//   (this object) <-> Device 1 (EtherCAT)/Term 1 (EK1200)/Term 5 (EK1122)/EK1100_ST1K2_ZOS/ST1K1-EL5042
//     Enc/Inputs/In/nComState @bit 1 <-> WcState/InputToggle
//     Enc/Inputs/In/nComState <-> WcState/WcState
//     Enc/Inputs/In/nDataIn1 <-> FB Inputs Channel 1/Position
//     Enc/Inputs/In/nState1 @bit 12 <-> FB Inputs Channel 1/Status/Diag
//     Enc/Inputs/In/nState1 @bit 1 <-> FB Inputs Channel 1/Status/Error
//     Enc/Inputs/In/nState1 @bit 14 <-> FB Inputs Channel 1/Status/Input cycle counter
//     Enc/Inputs/In/nState1 @bit 2 <-> FB Inputs Channel 1/Status/Ready
//     Enc/Inputs/In/nState1 @bit 13 <-> FB Inputs Channel 1/Status/TxPDO State
//     Enc/Inputs/In/nState1 <-> FB Inputs Channel 1/Status/Warning
//   (this object) <-> Device 1 (EtherCAT)/Term 1 (EK1200)/Term 5 (EK1122)/EK1100_ST1K2_ZOS/ST1K1-EL7041
//     Drive/Inputs/In/nState1 @bit 3 <-> STM Status/Status/Error
//     Drive/Inputs/In/nState1 @bit 5 <-> STM Status/Status/Moving negative
//     Drive/Inputs/In/nState1 @bit 4 <-> STM Status/Status/Moving positive
//     Drive/Inputs/In/nState1 @bit 1 <-> STM Status/Status/Ready
//     Drive/Inputs/In/nState1 <-> STM Status/Status/Ready to enable
//     Drive/Inputs/In/nState1 @bit 6 <-> STM Status/Status/Torque reduced
//     Drive/Inputs/In/nState1 @bit 2 <-> STM Status/Status/Warning
//     Drive/Inputs/In/nState2 @bit 3 <-> STM Status/Status/Digital input 1
//     Drive/Inputs/In/nState2 @bit 4 <-> STM Status/Status/Digital input 2
//     Drive/Inputs/In/nState2 @bit 5 <-> STM Status/Status/Sync error
//     Drive/Inputs/In/nState2 @bit 7 <-> STM Status/Status/TxPDO Toggle
//     Drive/Inputs/In/nState4 @bit 1 <-> WcState/InputToggle
//     Drive/Inputs/In/nState4 <-> WcState/WcState
//     Drive/Outputs/Out/nCtrl1 <-> STM Control/Control/Enable
//     Drive/Outputs/Out/nCtrl1 @bit 2 <-> STM Control/Control/Reduce torque
//     Drive/Outputs/Out/nCtrl1 @bit 1 <-> STM Control/Control/Reset
//     Drive/Outputs/Out/nDataOut2[0] <-> STM Velocity/Velocity
//   (this object) <-> Device 1 (EtherCAT)/Term 1 (EK1200)/Term 79 (EK1521-0010)/Term 306 (EK1501-0010)/Term 310 (EK1122)/EK1100_MR2K2/EL5042_M2K2X_M2K2Y
//     Enc/Inputs/In/nComState @bit 1 <-> WcState/InputToggle
//     Enc/Inputs/In/nComState <-> WcState/WcState
//     Enc/Inputs/In/nDataIn1 <-> FB Inputs Channel 1/Position
//     Enc/Inputs/In/nDataIn1 <-> FB Inputs Channel 2/Position
//     Enc/Inputs/In/nState1 @bit 12 <-> FB Inputs Channel 1/Status/Diag
//     Enc/Inputs/In/nState1 @bit 12 <-> FB Inputs Channel 2/Status/Diag
//     Enc/Inputs/In/nState1 @bit 1 <-> FB Inputs Channel 1/Status/Error
//     Enc/Inputs/In/nState1 @bit 1 <-> FB Inputs Channel 2/Status/Error
//     Enc/Inputs/In/nState1 @bit 14 <-> FB Inputs Channel 1/Status/Input cycle counter
//     Enc/Inputs/In/nState1 @bit 14 <-> FB Inputs Channel 2/Status/Input cycle counter
//     Enc/Inputs/In/nState1 @bit 2 <-> FB Inputs Channel 1/Status/Ready
//     Enc/Inputs/In/nState1 @bit 2 <-> FB Inputs Channel 2/Status/Ready
//     Enc/Inputs/In/nState1 @bit 13 <-> FB Inputs Channel 1/Status/TxPDO State
//     Enc/Inputs/In/nState1 @bit 13 <-> FB Inputs Channel 2/Status/TxPDO State
//     Enc/Inputs/In/nState1 <-> FB Inputs Channel 1/Status/Warning
//     Enc/Inputs/In/nState1 <-> FB Inputs Channel 2/Status/Warning
//   (this object) <-> Device 1 (EtherCAT)/Term 1 (EK1200)/Term 79 (EK1521-0010)/Term 306 (EK1501-0010)/Term 310 (EK1122)/EK1100_MR2K2/EL7041_M2K2X
//     Drive/Inputs/In/nState1 @bit 3 <-> STM Status/Status/Error
//     Drive/Inputs/In/nState1 @bit 5 <-> STM Status/Status/Moving negative
//     Drive/Inputs/In/nState1 @bit 4 <-> STM Status/Status/Moving positive
//     Drive/Inputs/In/nState1 @bit 1 <-> STM Status/Status/Ready
//     Drive/Inputs/In/nState1 <-> STM Status/Status/Ready to enable
//     Drive/Inputs/In/nState1 @bit 6 <-> STM Status/Status/Torque reduced
//     Drive/Inputs/In/nState1 @bit 2 <-> STM Status/Status/Warning
//     Drive/Inputs/In/nState2 @bit 3 <-> STM Status/Status/Digital input 1
//     Drive/Inputs/In/nState2 @bit 4 <-> STM Status/Status/Digital input 2
//     Drive/Inputs/In/nState2 @bit 5 <-> STM Status/Status/Sync error
//     Drive/Inputs/In/nState2 @bit 7 <-> STM Status/Status/TxPDO Toggle
//     Drive/Inputs/In/nState4 @bit 1 <-> WcState/InputToggle
//     Drive/Inputs/In/nState4 <-> WcState/WcState
//     Drive/Outputs/Out/nCtrl1 <-> STM Control/Control/Enable
//     Drive/Outputs/Out/nCtrl1 @bit 2 <-> STM Control/Control/Reduce torque
//     Drive/Outputs/Out/nCtrl1 @bit 1 <-> STM Control/Control/Reset
//     Drive/Outputs/Out/nDataOut2[0] <-> STM Velocity/Velocity
//   (this object) <-> Device 1 (EtherCAT)/Term 1 (EK1200)/Term 79 (EK1521-0010)/Term 306 (EK1501-0010)/Term 310 (EK1122)/EK1100_MR2K2/EL7041_M2K2Y
//     Drive/Inputs/In/nState1 @bit 3 <-> STM Status/Status/Error
//     Drive/Inputs/In/nState1 @bit 5 <-> STM Status/Status/Moving negative
//     Drive/Inputs/In/nState1 @bit 4 <-> STM Status/Status/Moving positive
//     Drive/Inputs/In/nState1 @bit 1 <-> STM Status/Status/Ready
//     Drive/Inputs/In/nState1 <-> STM Status/Status/Ready to enable
//     Drive/Inputs/In/nState1 @bit 6 <-> STM Status/Status/Torque reduced
//     Drive/Inputs/In/nState1 @bit 2 <-> STM Status/Status/Warning
//     Drive/Inputs/In/nState2 @bit 3 <-> STM Status/Status/Digital input 1
//     Drive/Inputs/In/nState2 @bit 4 <-> STM Status/Status/Digital input 2
//     Drive/Inputs/In/nState2 @bit 5 <-> STM Status/Status/Sync error
//     Drive/Inputs/In/nState2 @bit 7 <-> STM Status/Status/TxPDO Toggle
//     Drive/Inputs/In/nState4 @bit 1 <-> WcState/InputToggle
//     Drive/Inputs/In/nState4 <-> WcState/WcState
//     Drive/Outputs/Out/nCtrl1 <-> STM Control/Control/Enable
//     Drive/Outputs/Out/nCtrl1 @bit 2 <-> STM Control/Control/Reduce torque
//     Drive/Outputs/Out/nCtrl1 @bit 1 <-> STM Control/Control/Reset
//     Drive/Outputs/Out/nDataOut2[0] <-> STM Velocity/Velocity
//   (this object) <-> Device 1 (EtherCAT)/Term 1 (EK1200)/Term 79 (EK1521-0010)/Term 306 (EK1501-0010)/Term 310 (EK1122)/EK1100_MR2K2/EL5042_M2K2rX
//     Enc/Inputs/In/nComState @bit 1 <-> WcState/InputToggle
//     Enc/Inputs/In/nComState <-> WcState/WcState
//     Enc/Inputs/In/nDataIn1 <-> FB Inputs Channel 1/Position
//     Enc/Inputs/In/nState1 @bit 12 <-> FB Inputs Channel 1/Status/Diag
//     Enc/Inputs/In/nState1 @bit 1 <-> FB Inputs Channel 1/Status/Error
//     Enc/Inputs/In/nState1 @bit 14 <-> FB Inputs Channel 1/Status/Input cycle counter
//     Enc/Inputs/In/nState1 @bit 2 <-> FB Inputs Channel 1/Status/Ready
//     Enc/Inputs/In/nState1 @bit 13 <-> FB Inputs Channel 1/Status/TxPDO State
//     Enc/Inputs/In/nState1 <-> FB Inputs Channel 1/Status/Warning
//   (this object) <-> Device 1 (EtherCAT)/Term 1 (EK1200)/Term 79 (EK1521-0010)/Term 306 (EK1501-0010)/Term 310 (EK1122)/EK1100_MR2K2/EL7041_M2K2rX
//     Drive/Inputs/In/nState1 @bit 3 <-> STM Status/Status/Error
//     Drive/Inputs/In/nState1 @bit 5 <-> STM Status/Status/Moving negative
//     Drive/Inputs/In/nState1 @bit 4 <-> STM Status/Status/Moving positive
//     Drive/Inputs/In/nState1 @bit 1 <-> STM Status/Status/Ready
//     Drive/Inputs/In/nState1 <-> STM Status/Status/Ready to enable
//     Drive/Inputs/In/nState1 @bit 6 <-> STM Status/Status/Torque reduced
//     Drive/Inputs/In/nState1 @bit 2 <-> STM Status/Status/Warning
//     Drive/Inputs/In/nState2 @bit 3 <-> STM Status/Status/Digital input 1
//     Drive/Inputs/In/nState2 @bit 4 <-> STM Status/Status/Digital input 2
//     Drive/Inputs/In/nState2 @bit 5 <-> STM Status/Status/Sync error
//     Drive/Inputs/In/nState2 @bit 7 <-> STM Status/Status/TxPDO Toggle
//     Drive/Inputs/In/nState4 @bit 1 <-> WcState/InputToggle
//     Drive/Inputs/In/nState4 <-> WcState/WcState
//     Drive/Outputs/Out/nCtrl1 <-> STM Control/Control/Enable
//     Drive/Outputs/Out/nCtrl1 @bit 2 <-> STM Control/Control/Reduce torque
//     Drive/Outputs/Out/nCtrl1 @bit 1 <-> STM Control/Control/Reset
//     Drive/Outputs/Out/nDataOut2[0] <-> STM Velocity/Velocity
//   (this object) <-> Device 1 (EtherCAT)/Term 1 (EK1200)/Term 79 (EK1521-0010)/Term 306 (EK1501-0010)/Term 310 (EK1122)/EK1100_MR3K2/EL5042_M3K2X_M3K2Y
//     Enc/Inputs/In/nComState @bit 1 <-> WcState/InputToggle
//     Enc/Inputs/In/nComState <-> WcState/WcState
//     Enc/Inputs/In/nDataIn1 <-> FB Inputs Channel 1/Position
//     Enc/Inputs/In/nDataIn1 <-> FB Inputs Channel 2/Position
//     Enc/Inputs/In/nState1 @bit 12 <-> FB Inputs Channel 1/Status/Diag
//     Enc/Inputs/In/nState1 @bit 12 <-> FB Inputs Channel 2/Status/Diag
//     Enc/Inputs/In/nState1 @bit 1 <-> FB Inputs Channel 1/Status/Error
//     Enc/Inputs/In/nState1 @bit 1 <-> FB Inputs Channel 2/Status/Error
//     Enc/Inputs/In/nState1 @bit 14 <-> FB Inputs Channel 1/Status/Input cycle counter
//     Enc/Inputs/In/nState1 @bit 14 <-> FB Inputs Channel 2/Status/Input cycle counter
//     Enc/Inputs/In/nState1 @bit 2 <-> FB Inputs Channel 1/Status/Ready
//     Enc/Inputs/In/nState1 @bit 2 <-> FB Inputs Channel 2/Status/Ready
//     Enc/Inputs/In/nState1 @bit 13 <-> FB Inputs Channel 1/Status/TxPDO State
//     Enc/Inputs/In/nState1 @bit 13 <-> FB Inputs Channel 2/Status/TxPDO State
//     Enc/Inputs/In/nState1 <-> FB Inputs Channel 1/Status/Warning
//     Enc/Inputs/In/nState1 <-> FB Inputs Channel 2/Status/Warning
//   (this object) <-> Device 1 (EtherCAT)/Term 1 (EK1200)/Term 79 (EK1521-0010)/Term 306 (EK1501-0010)/Term 310 (EK1122)/EK1100_MR3K2/EL7041_M3K2X
//     Drive/Inputs/In/nState1 @bit 3 <-> STM Status/Status/Error
//     Drive/Inputs/In/nState1 @bit 5 <-> STM Status/Status/Moving negative
//     Drive/Inputs/In/nState1 @bit 4 <-> STM Status/Status/Moving positive
//     Drive/Inputs/In/nState1 @bit 1 <-> STM Status/Status/Ready
//     Drive/Inputs/In/nState1 <-> STM Status/Status/Ready to enable
//     Drive/Inputs/In/nState1 @bit 6 <-> STM Status/Status/Torque reduced
//     Drive/Inputs/In/nState1 @bit 2 <-> STM Status/Status/Warning
//     Drive/Inputs/In/nState2 @bit 3 <-> STM Status/Status/Digital input 1
//     Drive/Inputs/In/nState2 @bit 4 <-> STM Status/Status/Digital input 2
//     Drive/Inputs/In/nState2 @bit 5 <-> STM Status/Status/Sync error
//     Drive/Inputs/In/nState2 @bit 7 <-> STM Status/Status/TxPDO Toggle
//     Drive/Inputs/In/nState4 @bit 1 <-> WcState/InputToggle
//     Drive/Inputs/In/nState4 <-> WcState/WcState
//     Drive/Outputs/Out/nCtrl1 <-> STM Control/Control/Enable
//     Drive/Outputs/Out/nCtrl1 @bit 2 <-> STM Control/Control/Reduce torque
//     Drive/Outputs/Out/nCtrl1 @bit 1 <-> STM Control/Control/Reset
//     Drive/Outputs/Out/nDataOut2[0] <-> STM Velocity/Velocity
//   (this object) <-> Device 1 (EtherCAT)/Term 1 (EK1200)/Term 79 (EK1521-0010)/Term 306 (EK1501-0010)/Term 310 (EK1122)/EK1100_MR3K2/EL7041_M3K2Y
//     Drive/Inputs/In/nState1 @bit 3 <-> STM Status/Status/Error
//     Drive/Inputs/In/nState1 @bit 5 <-> STM Status/Status/Moving negative
//     Drive/Inputs/In/nState1 @bit 4 <-> STM Status/Status/Moving positive
//     Drive/Inputs/In/nState1 @bit 1 <-> STM Status/Status/Ready
//     Drive/Inputs/In/nState1 <-> STM Status/Status/Ready to enable
//     Drive/Inputs/In/nState1 @bit 6 <-> STM Status/Status/Torque reduced
//     Drive/Inputs/In/nState1 @bit 2 <-> STM Status/Status/Warning
//     Drive/Inputs/In/nState2 @bit 3 <-> STM Status/Status/Digital input 1
//     Drive/Inputs/In/nState2 @bit 4 <-> STM Status/Status/Digital input 2
//     Drive/Inputs/In/nState2 @bit 5 <-> STM Status/Status/Sync error
//     Drive/Inputs/In/nState2 @bit 7 <-> STM Status/Status/TxPDO Toggle
//     Drive/Inputs/In/nState4 @bit 1 <-> WcState/InputToggle
//     Drive/Inputs/In/nState4 <-> WcState/WcState
//     Drive/Outputs/Out/nCtrl1 <-> STM Control/Control/Enable
//     Drive/Outputs/Out/nCtrl1 @bit 2 <-> STM Control/Control/Reduce torque
//     Drive/Outputs/Out/nCtrl1 @bit 1 <-> STM Control/Control/Reset
//     Drive/Outputs/Out/nDataOut2[0] <-> STM Velocity/Velocity
//   (this object) <-> Device 1 (EtherCAT)/Term 1 (EK1200)/Term 79 (EK1521-0010)/Term 306 (EK1501-0010)/Term 310 (EK1122)/EK1100_MR3K2/EL5042_M3K2rY
//     Enc/Inputs/In/nComState @bit 1 <-> WcState/InputToggle
//     Enc/Inputs/In/nComState <-> WcState/WcState
//     Enc/Inputs/In/nDataIn1 <-> FB Inputs Channel 1/Position
//     Enc/Inputs/In/nState1 @bit 12 <-> FB Inputs Channel 1/Status/Diag
//     Enc/Inputs/In/nState1 @bit 1 <-> FB Inputs Channel 1/Status/Error
//     Enc/Inputs/In/nState1 @bit 14 <-> FB Inputs Channel 1/Status/Input cycle counter
//     Enc/Inputs/In/nState1 @bit 2 <-> FB Inputs Channel 1/Status/Ready
//     Enc/Inputs/In/nState1 @bit 13 <-> FB Inputs Channel 1/Status/TxPDO State
//     Enc/Inputs/In/nState1 <-> FB Inputs Channel 1/Status/Warning
//   (this object) <-> Device 1 (EtherCAT)/Term 1 (EK1200)/Term 79 (EK1521-0010)/Term 306 (EK1501-0010)/Term 310 (EK1122)/EK1100_MR3K2/EL7041_M3K2rY
//     Drive/Inputs/In/nState1 @bit 3 <-> STM Status/Status/Error
//     Drive/Inputs/In/nState1 @bit 5 <-> STM Status/Status/Moving negative
//     Drive/Inputs/In/nState1 @bit 4 <-> STM Status/Status/Moving positive
//     Drive/Inputs/In/nState1 @bit 1 <-> STM Status/Status/Ready
//     Drive/Inputs/In/nState1 <-> STM Status/Status/Ready to enable
//     Drive/Inputs/In/nState1 @bit 6 <-> STM Status/Status/Torque reduced
//     Drive/Inputs/In/nState1 @bit 2 <-> STM Status/Status/Warning
//     Drive/Inputs/In/nState2 @bit 3 <-> STM Status/Status/Digital input 1
//     Drive/Inputs/In/nState2 @bit 4 <-> STM Status/Status/Digital input 2
//     Drive/Inputs/In/nState2 @bit 5 <-> STM Status/Status/Sync error
//     Drive/Inputs/In/nState2 @bit 7 <-> STM Status/Status/TxPDO Toggle
//     Drive/Inputs/In/nState4 @bit 1 <-> WcState/InputToggle
//     Drive/Inputs/In/nState4 <-> WcState/WcState
//     Drive/Outputs/Out/nCtrl1 <-> STM Control/Control/Enable
//     Drive/Outputs/Out/nCtrl1 @bit 2 <-> STM Control/Control/Reduce torque
//     Drive/Outputs/Out/nCtrl1 @bit 1 <-> STM Control/Control/Reset
//     Drive/Outputs/Out/nDataOut2[0] <-> STM Velocity/Velocity
//   (this object) <-> Device 1 (EtherCAT)/Term 1 (EK1200)/Term 79 (EK1521-0010)/Term 306 (EK1501-0010)/Term 310 (EK1122)/EK1100_MR3K2_BENDER/EL5042_M3K2_BEND_USDS
//     Enc/Inputs/In/nComState @bit 1 <-> WcState/InputToggle
//     Enc/Inputs/In/nComState <-> WcState/WcState
//     Enc/Inputs/In/nDataIn1 <-> FB Inputs Channel 1/Position
//     Enc/Inputs/In/nDataIn1 <-> FB Inputs Channel 2/Position
//     Enc/Inputs/In/nState1 @bit 12 <-> FB Inputs Channel 1/Status/Diag
//     Enc/Inputs/In/nState1 @bit 12 <-> FB Inputs Channel 2/Status/Diag
//     Enc/Inputs/In/nState1 @bit 1 <-> FB Inputs Channel 1/Status/Error
//     Enc/Inputs/In/nState1 @bit 1 <-> FB Inputs Channel 2/Status/Error
//     Enc/Inputs/In/nState1 @bit 14 <-> FB Inputs Channel 1/Status/Input cycle counter
//     Enc/Inputs/In/nState1 @bit 14 <-> FB Inputs Channel 2/Status/Input cycle counter
//     Enc/Inputs/In/nState1 @bit 2 <-> FB Inputs Channel 1/Status/Ready
//     Enc/Inputs/In/nState1 @bit 2 <-> FB Inputs Channel 2/Status/Ready
//     Enc/Inputs/In/nState1 @bit 13 <-> FB Inputs Channel 1/Status/TxPDO State
//     Enc/Inputs/In/nState1 @bit 13 <-> FB Inputs Channel 2/Status/TxPDO State
//     Enc/Inputs/In/nState1 <-> FB Inputs Channel 1/Status/Warning
//     Enc/Inputs/In/nState1 <-> FB Inputs Channel 2/Status/Warning
//   (this object) <-> Device 1 (EtherCAT)/Term 1 (EK1200)/Term 79 (EK1521-0010)/Term 306 (EK1501-0010)/Term 310 (EK1122)/EK1100_MR3K2_BENDER/EL7041_M3K2_BEND_US
//     Drive/Inputs/In/nState1 @bit 3 <-> STM Status/Status/Error
//     Drive/Inputs/In/nState1 @bit 5 <-> STM Status/Status/Moving negative
//     Drive/Inputs/In/nState1 @bit 4 <-> STM Status/Status/Moving positive
//     Drive/Inputs/In/nState1 @bit 1 <-> STM Status/Status/Ready
//     Drive/Inputs/In/nState1 <-> STM Status/Status/Ready to enable
//     Drive/Inputs/In/nState1 @bit 6 <-> STM Status/Status/Torque reduced
//     Drive/Inputs/In/nState1 @bit 2 <-> STM Status/Status/Warning
//     Drive/Inputs/In/nState2 @bit 3 <-> STM Status/Status/Digital input 1
//     Drive/Inputs/In/nState2 @bit 4 <-> STM Status/Status/Digital input 2
//     Drive/Inputs/In/nState2 @bit 5 <-> STM Status/Status/Sync error
//     Drive/Inputs/In/nState2 @bit 7 <-> STM Status/Status/TxPDO Toggle
//     Drive/Inputs/In/nState4 @bit 1 <-> WcState/InputToggle
//     Drive/Inputs/In/nState4 <-> WcState/WcState
//     Drive/Outputs/Out/nCtrl1 <-> STM Control/Control/Enable
//     Drive/Outputs/Out/nCtrl1 @bit 2 <-> STM Control/Control/Reduce torque
//     Drive/Outputs/Out/nCtrl1 @bit 1 <-> STM Control/Control/Reset
//     Drive/Outputs/Out/nDataOut2[0] <-> STM Velocity/Velocity
//   (this object) <-> Device 1 (EtherCAT)/Term 1 (EK1200)/Term 79 (EK1521-0010)/Term 306 (EK1501-0010)/Term 310 (EK1122)/EK1100_MR3K2_BENDER/EL7041_M3K2_BEND_DS
//     Drive/Inputs/In/nState1 @bit 3 <-> STM Status/Status/Error
//     Drive/Inputs/In/nState1 @bit 5 <-> STM Status/Status/Moving negative
//     Drive/Inputs/In/nState1 @bit 4 <-> STM Status/Status/Moving positive
//     Drive/Inputs/In/nState1 @bit 1 <-> STM Status/Status/Ready
//     Drive/Inputs/In/nState1 <-> STM Status/Status/Ready to enable
//     Drive/Inputs/In/nState1 @bit 6 <-> STM Status/Status/Torque reduced
//     Drive/Inputs/In/nState1 @bit 2 <-> STM Status/Status/Warning
//     Drive/Inputs/In/nState2 @bit 3 <-> STM Status/Status/Digital input 1
//     Drive/Inputs/In/nState2 @bit 4 <-> STM Status/Status/Digital input 2
//     Drive/Inputs/In/nState2 @bit 5 <-> STM Status/Status/Sync error
//     Drive/Inputs/In/nState2 @bit 7 <-> STM Status/Status/TxPDO Toggle
//     Drive/Inputs/In/nState4 @bit 1 <-> WcState/InputToggle
//     Drive/Inputs/In/nState4 <-> WcState/WcState
//     Drive/Outputs/Out/nCtrl1 <-> STM Control/Control/Enable
//     Drive/Outputs/Out/nCtrl1 @bit 2 <-> STM Control/Control/Reduce torque
//     Drive/Outputs/Out/nCtrl1 @bit 1 <-> STM Control/Control/Reset
//     Drive/Outputs/Out/nDataOut2[0] <-> STM Velocity/Velocity
//   (this object) <-> Device 1 (EtherCAT)/Term 1 (EK1200)/Term 79 (EK1521-0010)/Term 306 (EK1501-0010)/Term 322 (EK1122)/EK1100_MR4K2/EL5042_M4K2X_M4K2Y
//     Enc/Inputs/In/nComState @bit 1 <-> WcState/InputToggle
//     Enc/Inputs/In/nComState <-> WcState/WcState
//     Enc/Inputs/In/nDataIn1 <-> FB Inputs Channel 1/Position
//     Enc/Inputs/In/nDataIn1 <-> FB Inputs Channel 2/Position
//     Enc/Inputs/In/nState1 @bit 12 <-> FB Inputs Channel 1/Status/Diag
//     Enc/Inputs/In/nState1 @bit 12 <-> FB Inputs Channel 2/Status/Diag
//     Enc/Inputs/In/nState1 @bit 1 <-> FB Inputs Channel 1/Status/Error
//     Enc/Inputs/In/nState1 @bit 1 <-> FB Inputs Channel 2/Status/Error
//     Enc/Inputs/In/nState1 @bit 14 <-> FB Inputs Channel 1/Status/Input cycle counter
//     Enc/Inputs/In/nState1 @bit 14 <-> FB Inputs Channel 2/Status/Input cycle counter
//     Enc/Inputs/In/nState1 @bit 2 <-> FB Inputs Channel 1/Status/Ready
//     Enc/Inputs/In/nState1 @bit 2 <-> FB Inputs Channel 2/Status/Ready
//     Enc/Inputs/In/nState1 @bit 13 <-> FB Inputs Channel 1/Status/TxPDO State
//     Enc/Inputs/In/nState1 @bit 13 <-> FB Inputs Channel 2/Status/TxPDO State
//     Enc/Inputs/In/nState1 <-> FB Inputs Channel 1/Status/Warning
//     Enc/Inputs/In/nState1 <-> FB Inputs Channel 2/Status/Warning
//   (this object) <-> Device 1 (EtherCAT)/Term 1 (EK1200)/Term 79 (EK1521-0010)/Term 306 (EK1501-0010)/Term 322 (EK1122)/EK1100_MR4K2/EL7041_M4K2X
//     Drive/Inputs/In/nState1 @bit 3 <-> STM Status/Status/Error
//     Drive/Inputs/In/nState1 @bit 5 <-> STM Status/Status/Moving negative
//     Drive/Inputs/In/nState1 @bit 4 <-> STM Status/Status/Moving positive
//     Drive/Inputs/In/nState1 @bit 1 <-> STM Status/Status/Ready
//     Drive/Inputs/In/nState1 <-> STM Status/Status/Ready to enable
//     Drive/Inputs/In/nState1 @bit 6 <-> STM Status/Status/Torque reduced
//     Drive/Inputs/In/nState1 @bit 2 <-> STM Status/Status/Warning
//     Drive/Inputs/In/nState2 @bit 3 <-> STM Status/Status/Digital input 1
//     Drive/Inputs/In/nState2 @bit 4 <-> STM Status/Status/Digital input 2
//     Drive/Inputs/In/nState2 @bit 5 <-> STM Status/Status/Sync error
//     Drive/Inputs/In/nState2 @bit 7 <-> STM Status/Status/TxPDO Toggle
//     Drive/Inputs/In/nState4 @bit 1 <-> WcState/InputToggle
//     Drive/Inputs/In/nState4 <-> WcState/WcState
//     Drive/Outputs/Out/nCtrl1 <-> STM Control/Control/Enable
//     Drive/Outputs/Out/nCtrl1 @bit 2 <-> STM Control/Control/Reduce torque
//     Drive/Outputs/Out/nCtrl1 @bit 1 <-> STM Control/Control/Reset
//     Drive/Outputs/Out/nDataOut2[0] <-> STM Velocity/Velocity
//   (this object) <-> Device 1 (EtherCAT)/Term 1 (EK1200)/Term 79 (EK1521-0010)/Term 306 (EK1501-0010)/Term 322 (EK1122)/EK1100_MR4K2/EL7041_M4K2Y
//     Drive/Inputs/In/nState1 @bit 3 <-> STM Status/Status/Error
//     Drive/Inputs/In/nState1 @bit 5 <-> STM Status/Status/Moving negative
//     Drive/Inputs/In/nState1 @bit 4 <-> STM Status/Status/Moving positive
//     Drive/Inputs/In/nState1 @bit 1 <-> STM Status/Status/Ready
//     Drive/Inputs/In/nState1 <-> STM Status/Status/Ready to enable
//     Drive/Inputs/In/nState1 @bit 6 <-> STM Status/Status/Torque reduced
//     Drive/Inputs/In/nState1 @bit 2 <-> STM Status/Status/Warning
//     Drive/Inputs/In/nState2 @bit 3 <-> STM Status/Status/Digital input 1
//     Drive/Inputs/In/nState2 @bit 4 <-> STM Status/Status/Digital input 2
//     Drive/Inputs/In/nState2 @bit 5 <-> STM Status/Status/Sync error
//     Drive/Inputs/In/nState2 @bit 7 <-> STM Status/Status/TxPDO Toggle
//     Drive/Inputs/In/nState4 @bit 1 <-> WcState/InputToggle
//     Drive/Inputs/In/nState4 <-> WcState/WcState
//     Drive/Outputs/Out/nCtrl1 <-> STM Control/Control/Enable
//     Drive/Outputs/Out/nCtrl1 @bit 2 <-> STM Control/Control/Reduce torque
//     Drive/Outputs/Out/nCtrl1 @bit 1 <-> STM Control/Control/Reset
//     Drive/Outputs/Out/nDataOut2[0] <-> STM Velocity/Velocity
//   (this object) <-> Device 1 (EtherCAT)/Term 1 (EK1200)/Term 79 (EK1521-0010)/Term 306 (EK1501-0010)/Term 322 (EK1122)/EK1100_MR4K2/EL5042_M4K2rX
//     Enc/Inputs/In/nComState @bit 1 <-> WcState/InputToggle
//     Enc/Inputs/In/nComState <-> WcState/WcState
//     Enc/Inputs/In/nDataIn1 <-> FB Inputs Channel 1/Position
//     Enc/Inputs/In/nState1 @bit 12 <-> FB Inputs Channel 1/Status/Diag
//     Enc/Inputs/In/nState1 @bit 1 <-> FB Inputs Channel 1/Status/Error
//     Enc/Inputs/In/nState1 @bit 14 <-> FB Inputs Channel 1/Status/Input cycle counter
//     Enc/Inputs/In/nState1 @bit 2 <-> FB Inputs Channel 1/Status/Ready
//     Enc/Inputs/In/nState1 @bit 13 <-> FB Inputs Channel 1/Status/TxPDO State
//     Enc/Inputs/In/nState1 <-> FB Inputs Channel 1/Status/Warning
//   (this object) <-> Device 1 (EtherCAT)/Term 1 (EK1200)/Term 79 (EK1521-0010)/Term 306 (EK1501-0010)/Term 322 (EK1122)/EK1100_MR4K2/EL7041_M4K2rX
//     Drive/Inputs/In/nState1 @bit 3 <-> STM Status/Status/Error
//     Drive/Inputs/In/nState1 @bit 5 <-> STM Status/Status/Moving negative
//     Drive/Inputs/In/nState1 @bit 4 <-> STM Status/Status/Moving positive
//     Drive/Inputs/In/nState1 @bit 1 <-> STM Status/Status/Ready
//     Drive/Inputs/In/nState1 <-> STM Status/Status/Ready to enable
//     Drive/Inputs/In/nState1 @bit 6 <-> STM Status/Status/Torque reduced
//     Drive/Inputs/In/nState1 @bit 2 <-> STM Status/Status/Warning
//     Drive/Inputs/In/nState2 @bit 3 <-> STM Status/Status/Digital input 1
//     Drive/Inputs/In/nState2 @bit 4 <-> STM Status/Status/Digital input 2
//     Drive/Inputs/In/nState2 @bit 5 <-> STM Status/Status/Sync error
//     Drive/Inputs/In/nState2 @bit 7 <-> STM Status/Status/TxPDO Toggle
//     Drive/Inputs/In/nState4 @bit 1 <-> WcState/InputToggle
//     Drive/Inputs/In/nState4 <-> WcState/WcState
//     Drive/Outputs/Out/nCtrl1 <-> STM Control/Control/Enable
//     Drive/Outputs/Out/nCtrl1 @bit 2 <-> STM Control/Control/Reduce torque
//     Drive/Outputs/Out/nCtrl1 @bit 1 <-> STM Control/Control/Reset
//     Drive/Outputs/Out/nDataOut2[0] <-> STM Velocity/Velocity
//   (this object) <-> Device 1 (EtherCAT)/Term 1 (EK1200)/Term 79 (EK1521-0010)/Term 306 (EK1501-0010)/Term 322 (EK1122)/EK1100_MR4K2_BENDER/EL5042_M4K2_BEND_USDS
//     Enc/Inputs/In/nComState @bit 1 <-> WcState/InputToggle
//     Enc/Inputs/In/nComState <-> WcState/WcState
//     Enc/Inputs/In/nDataIn1 <-> FB Inputs Channel 1/Position
//     Enc/Inputs/In/nDataIn1 <-> FB Inputs Channel 2/Position
//     Enc/Inputs/In/nState1 @bit 12 <-> FB Inputs Channel 1/Status/Diag
//     Enc/Inputs/In/nState1 @bit 12 <-> FB Inputs Channel 2/Status/Diag
//     Enc/Inputs/In/nState1 @bit 1 <-> FB Inputs Channel 1/Status/Error
//     Enc/Inputs/In/nState1 @bit 1 <-> FB Inputs Channel 2/Status/Error
//     Enc/Inputs/In/nState1 @bit 14 <-> FB Inputs Channel 1/Status/Input cycle counter
//     Enc/Inputs/In/nState1 @bit 14 <-> FB Inputs Channel 2/Status/Input cycle counter
//     Enc/Inputs/In/nState1 @bit 2 <-> FB Inputs Channel 1/Status/Ready
//     Enc/Inputs/In/nState1 @bit 2 <-> FB Inputs Channel 2/Status/Ready
//     Enc/Inputs/In/nState1 @bit 13 <-> FB Inputs Channel 1/Status/TxPDO State
//     Enc/Inputs/In/nState1 @bit 13 <-> FB Inputs Channel 2/Status/TxPDO State
//     Enc/Inputs/In/nState1 <-> FB Inputs Channel 1/Status/Warning
//     Enc/Inputs/In/nState1 <-> FB Inputs Channel 2/Status/Warning
//   (this object) <-> Device 1 (EtherCAT)/Term 1 (EK1200)/Term 79 (EK1521-0010)/Term 306 (EK1501-0010)/Term 322 (EK1122)/EK1100_MR4K2_BENDER/EL7041_M4K2_BEND_US
//     Drive/Inputs/In/nState1 @bit 3 <-> STM Status/Status/Error
//     Drive/Inputs/In/nState1 @bit 5 <-> STM Status/Status/Moving negative
//     Drive/Inputs/In/nState1 @bit 4 <-> STM Status/Status/Moving positive
//     Drive/Inputs/In/nState1 @bit 1 <-> STM Status/Status/Ready
//     Drive/Inputs/In/nState1 <-> STM Status/Status/Ready to enable
//     Drive/Inputs/In/nState1 @bit 6 <-> STM Status/Status/Torque reduced
//     Drive/Inputs/In/nState1 @bit 2 <-> STM Status/Status/Warning
//     Drive/Inputs/In/nState2 @bit 3 <-> STM Status/Status/Digital input 1
//     Drive/Inputs/In/nState2 @bit 4 <-> STM Status/Status/Digital input 2
//     Drive/Inputs/In/nState2 @bit 5 <-> STM Status/Status/Sync error
//     Drive/Inputs/In/nState2 @bit 7 <-> STM Status/Status/TxPDO Toggle
//     Drive/Inputs/In/nState4 @bit 1 <-> WcState/InputToggle
//     Drive/Inputs/In/nState4 <-> WcState/WcState
//     Drive/Outputs/Out/nCtrl1 <-> STM Control/Control/Enable
//     Drive/Outputs/Out/nCtrl1 @bit 2 <-> STM Control/Control/Reduce torque
//     Drive/Outputs/Out/nCtrl1 @bit 1 <-> STM Control/Control/Reset
//     Drive/Outputs/Out/nDataOut2[0] <-> STM Velocity/Velocity
//   (this object) <-> Device 1 (EtherCAT)/Term 1 (EK1200)/Term 79 (EK1521-0010)/Term 306 (EK1501-0010)/Term 322 (EK1122)/EK1100_MR4K2_BENDER/EL7041_M4K2_BEND_DS
//     Drive/Inputs/In/nState1 @bit 3 <-> STM Status/Status/Error
//     Drive/Inputs/In/nState1 @bit 5 <-> STM Status/Status/Moving negative
//     Drive/Inputs/In/nState1 @bit 4 <-> STM Status/Status/Moving positive
//     Drive/Inputs/In/nState1 @bit 1 <-> STM Status/Status/Ready
//     Drive/Inputs/In/nState1 <-> STM Status/Status/Ready to enable
//     Drive/Inputs/In/nState1 @bit 6 <-> STM Status/Status/Torque reduced
//     Drive/Inputs/In/nState1 @bit 2 <-> STM Status/Status/Warning
//     Drive/Inputs/In/nState2 @bit 3 <-> STM Status/Status/Digital input 1
//     Drive/Inputs/In/nState2 @bit 4 <-> STM Status/Status/Digital input 2
//     Drive/Inputs/In/nState2 @bit 5 <-> STM Status/Status/Sync error
//     Drive/Inputs/In/nState2 @bit 7 <-> STM Status/Status/TxPDO Toggle
//     Drive/Inputs/In/nState4 @bit 1 <-> WcState/InputToggle
//     Drive/Inputs/In/nState4 <-> WcState/WcState
//     Drive/Outputs/Out/nCtrl1 <-> STM Control/Control/Enable
//     Drive/Outputs/Out/nCtrl1 @bit 2 <-> STM Control/Control/Reduce torque
//     Drive/Outputs/Out/nCtrl1 @bit 1 <-> STM Control/Control/Reset
//     Drive/Outputs/Out/nDataOut2[0] <-> STM Velocity/Velocity
//   rixs_optics Instance <-> Device 1 (EtherCAT)/Term 1 (EK1200)/E5 (EK1122)/Box 84 (EP2338-0002)
//     PlcTask Outputs/PRG_SP1K1_MONO.bLEDPower01 <-> Channel 10/Output
//     PlcTask Outputs/PRG_SP1K1_MONO.bLEDPower02 <-> Channel 12/Output
//     PlcTask Outputs/PRG_SP1K1_MONO.bLEDPower03 <-> Channel 14/Output
//   rixs_optics Instance <-> Device 1 (EtherCAT)/Term 1 (EK1200)/E5 (EK1122)/SL1K2-EXIT (EK1100)/EL2004_SL1K2
//     PlcTask Outputs/PRG_SL1K2_EXIT.bFanOn <-> Channel 1/Output
//     PlcTask Outputs/PRG_SL1K2_EXIT.bLEDPower <-> Channel 2/Output
//     PlcTask Outputs/PRG_SL1K2_EXIT.fbGige.bGigePower <-> Channel 3/Output
//   rixs_optics Instance <-> Device 1 (EtherCAT)/Term 1 (EK1200)/E5 (EK1122)/SL1K2-EXIT (EK1100)/EL3052_SL1K2_FWM
//     PlcTask Inputs/PRG_SL1K2_EXIT.fbFlowMeter.iRaw <-> AI Standard Channel 1/Value
//   rixs_optics Instance <-> Device 1 (EtherCAT)/Term 1 (EK1200)/E5 (EK1122)/SL1K2-EXIT (EK1100)/EL3201_SL1K2_1
//     PlcTask Inputs/PRG_SL1K2_EXIT.RTD_Crystal_TOP.bError <-> RTD/Status/Error
//     PlcTask Inputs/PRG_SL1K2_EXIT.RTD_Crystal_TOP.bOverrange <-> RTD/Status/Overrange
//     PlcTask Inputs/PRG_SL1K2_EXIT.RTD_Crystal_TOP.bUnderrange <-> RTD/Status/Underrange
//     PlcTask Inputs/PRG_SL1K2_EXIT.RTD_Crystal_TOP.iRaw <-> RTD/Value
//   rixs_optics Instance <-> Device 1 (EtherCAT)/Term 1 (EK1200)/E5 (EK1122)/SL1K2-EXIT (EK1100)/EL3201_SL1K2_2
//     PlcTask Inputs/PRG_SL1K2_EXIT.RTD_Crystal_BOTTOM.bError <-> RTD/Status/Error
//     PlcTask Inputs/PRG_SL1K2_EXIT.RTD_Crystal_BOTTOM.bOverrange <-> RTD/Status/Overrange
//     PlcTask Inputs/PRG_SL1K2_EXIT.RTD_Crystal_BOTTOM.bUnderrange <-> RTD/Status/Underrange
//     PlcTask Inputs/PRG_SL1K2_EXIT.RTD_Crystal_BOTTOM.iRaw <-> RTD/Value
//   rixs_optics Instance <-> Device 1 (EtherCAT)/Term 1 (EK1200)/E5 (EK1122)/SL1K2-EXIT (EK1100)/EL3201_SL1K2_3
//     PlcTask Inputs/PRG_SL1K2_EXIT.RTD_HeatSync.bError <-> RTD/Status/Error
//     PlcTask Inputs/PRG_SL1K2_EXIT.RTD_HeatSync.bOverrange <-> RTD/Status/Overrange
//     PlcTask Inputs/PRG_SL1K2_EXIT.RTD_HeatSync.bUnderrange <-> RTD/Status/Underrange
//     PlcTask Inputs/PRG_SL1K2_EXIT.RTD_HeatSync.iRaw <-> RTD/Value
//   rixs_optics Instance <-> Device 1 (EtherCAT)/Term 1 (EK1200)/E5 (EK1122)/SL1K2-EXIT (EK1100)/EL3201_SL1K2_4
//     PlcTask Inputs/PRG_SL1K2_EXIT.RTD_YAG.bError <-> RTD/Status/Error
//     PlcTask Inputs/PRG_SL1K2_EXIT.RTD_YAG.bOverrange <-> RTD/Status/Overrange
//     PlcTask Inputs/PRG_SL1K2_EXIT.RTD_YAG.bUnderrange <-> RTD/Status/Underrange
//     PlcTask Inputs/PRG_SL1K2_EXIT.RTD_YAG.iRaw <-> RTD/Value
//   rixs_optics Instance <-> Device 1 (EtherCAT)/Term 1 (EK1200)/E5 (EK1122)/SL1K2-EXIT (EK1100)/EL4004_SL1K2
//     PlcTask Outputs/PRG_SL1K2_EXIT.fbGige.iIlluminatorINT <-> AO Outputs Channel 1/Analog output
//   rixs_optics Instance <-> Device 1 (EtherCAT)/Term 1 (EK1200)/E5 (EK1122)/SL1K2-EXIT (EK1100)/EL5042_SL1K2_PITCH_VERT
//     PlcTask Inputs/Main.M19.nRawEncoderULINT <-> FB Inputs Channel 1/Position
//     PlcTask Inputs/Main.M20.nRawEncoderULINT <-> FB Inputs Channel 2/Position
//   rixs_optics Instance <-> Device 1 (EtherCAT)/Term 1 (EK1200)/E5 (EK1122)/SL1K2-EXIT (EK1100)/EL5042_SL1K2_ROLL_GAP
//     PlcTask Inputs/Main.M21.nRawEncoderULINT <-> FB Inputs Channel 1/Position
//     PlcTask Inputs/Main.M22.nRawEncoderULINT <-> FB Inputs Channel 2/Position
//   rixs_optics Instance <-> Device 1 (EtherCAT)/Term 1 (EK1200)/E5 (EK1122)/SL1K2-EXIT (EK1100)/EL5042_SL1K2_YAG
//     PlcTask Inputs/Main.M23.nRawEncoderULINT <-> FB Inputs Channel 1/Position
//   rixs_optics Instance <-> Device 1 (EtherCAT)/Term 1 (EK1200)/E5 (EK1122)/SL1K2-EXIT (EK1100)/EL7047_SL1K2_GAP
//     PlcTask Inputs/Main.M22.bLimitBackwardEnable <-> STM Status/Status/Digital input 2
//     PlcTask Inputs/Main.M22.bLimitForwardEnable <-> STM Status/Status/Digital input 1
//   rixs_optics Instance <-> Device 1 (EtherCAT)/Term 1 (EK1200)/E5 (EK1122)/SL1K2-EXIT (EK1100)/EL7047_SL1K2_PITCH
//     PlcTask Inputs/Main.M19.bLimitBackwardEnable <-> STM Status/Status/Digital input 1
//     PlcTask Inputs/Main.M19.bLimitForwardEnable <-> STM Status/Status/Digital input 2
//   rixs_optics Instance <-> Device 1 (EtherCAT)/Term 1 (EK1200)/E5 (EK1122)/SL1K2-EXIT (EK1100)/EL7047_SL1K2_ROLL
//     PlcTask Inputs/Main.M21.bLimitBackwardEnable <-> STM Status/Status/Digital input 1
//     PlcTask Inputs/Main.M21.bLimitForwardEnable <-> STM Status/Status/Digital input 2
//   rixs_optics Instance <-> Device 1 (EtherCAT)/Term 1 (EK1200)/E5 (EK1122)/SL1K2-EXIT (EK1100)/EL7047_SL1K2_VERT
//     PlcTask Inputs/Main.M20.bLimitBackwardEnable <-> STM Status/Status/Digital input 2
//     PlcTask Inputs/Main.M20.bLimitForwardEnable <-> STM Status/Status/Digital input 1
//   rixs_optics Instance <-> Device 1 (EtherCAT)/Term 1 (EK1200)/E5 (EK1122)/SL1K2-EXIT (EK1100)/EL7047_SL1K2_YAG
//     PlcTask Inputs/Main.M23.bLimitBackwardEnable <-> STM Status/Status/Digital input 1
//     PlcTask Inputs/Main.M23.bLimitForwardEnable <-> STM Status/Status/Digital input 2
//   rixs_optics Instance <-> Device 1 (EtherCAT)/Term 1 (EK1200)/E5 (EK1122)/SP1K1-EP3204-0002-EP2
//     PlcTask Inputs/PRG_SP1K1_MONO.RTD{1..4}.bError <-> RTD RTDInputs Channel {1..4}/Status/Error  (4 links)
//     PlcTask Inputs/PRG_SP1K1_MONO.RTD{1..4}.bOverrange <-> RTD RTDInputs Channel {1..4}/Status/Overrange  (4 links)
//     PlcTask Inputs/PRG_SP1K1_MONO.RTD{1..4}.bUnderrange <-> RTD RTDInputs Channel {1..4}/Status/Underrange  (4 links)
//     PlcTask Inputs/PRG_SP1K1_MONO.RTD{1..4}.iRaw <-> RTD RTDInputs Channel {1..4}/Value  (4 links)
//   rixs_optics Instance <-> Device 1 (EtherCAT)/Term 1 (EK1200)/E5 (EK1122)/X1 SP1K1-MONO(EK1100)/EL3054_SP1K1_FWM_PRSM
//     PlcTask Inputs/PRG_SP1K1_MONO.fSP1K1_Flow_1.iRaw <-> AI Standard Channel 1/Value
//     PlcTask Inputs/PRG_SP1K1_MONO.fSP1K1_Flow_2.iRaw <-> AI Standard Channel 2/Value
//     PlcTask Inputs/PRG_SP1K1_MONO.fSP1K1_Press_1.iRaw <-> AI Standard Channel 3/Value
//   rixs_optics Instance <-> Device 1 (EtherCAT)/Term 1 (EK1200)/E5 (EK1122)/X1 SP1K1-MONO(EK1100)/SP1K1-EL1004-E17
//     PlcTask Inputs/PRG_SP1K1_MONO.bSTOEnable1 <-> Channel 1/Input
//     PlcTask Inputs/PRG_SP1K1_MONO.bSTOEnable2 <-> Channel 2/Input
//   rixs_optics Instance <-> Device 1 (EtherCAT)/Term 1 (EK1200)/E5 (EK1122)/X1 SP1K1-MONO(EK1100)/SP1K1-EL3204-E15
//     PlcTask Inputs/PRG_SP1K1_MONO.RTD{5..8}.bError <-> RTD Inputs Channel {1..4}/Status/Error  (4 links)
//     PlcTask Inputs/PRG_SP1K1_MONO.RTD{5..8}.bOverrange <-> RTD Inputs Channel {1..4}/Status/Overrange  (4 links)
//     PlcTask Inputs/PRG_SP1K1_MONO.RTD{5..8}.bUnderrange <-> RTD Inputs Channel {1..4}/Status/Underrange  (4 links)
//     PlcTask Inputs/PRG_SP1K1_MONO.RTD{5..8}.iRaw <-> RTD Inputs Channel {1..4}/Value  (4 links)
//   rixs_optics Instance <-> Device 1 (EtherCAT)/Term 1 (EK1200)/E5 (EK1122)/X1 SP1K1-MONO(EK1100)/SP1K1-EL3204-E16
//     PlcTask Inputs/PRG_SP1K1_MONO.RTD{9..12}.bError <-> RTD Inputs Channel {1..4}/Status/Error  (4 links)
//     PlcTask Inputs/PRG_SP1K1_MONO.RTD{9..12}.bOverrange <-> RTD Inputs Channel {1..4}/Status/Overrange  (4 links)
//     PlcTask Inputs/PRG_SP1K1_MONO.RTD{9..12}.bUnderrange <-> RTD Inputs Channel {1..4}/Status/Underrange  (4 links)
//     PlcTask Inputs/PRG_SP1K1_MONO.RTD{9..12}.iRaw <-> RTD Inputs Channel {1..4}/Value  (4 links)
//   rixs_optics Instance <-> Device 1 (EtherCAT)/Term 1 (EK1200)/E5 (EK1122)/X1 SP1K1-MONO(EK1100)/g_h_m
//     PlcTask Inputs/Main.M9.bLimitBackwardEnable <-> STM Status/Status/Digital input 2
//     PlcTask Inputs/Main.M9.bLimitForwardEnable <-> STM Status/Status/Digital input 1
//   rixs_optics Instance <-> Device 1 (EtherCAT)/Term 1 (EK1200)/E5 (EK1122)/X1 SP1K1-MONO(EK1100)/g_pi_m
//     PlcTask Inputs/Main.M7.bLimitBackwardEnable <-> STM Status/Status/Digital input 2
//     PlcTask Inputs/Main.M7.bLimitForwardEnable <-> STM Status/Status/Digital input 1
//   rixs_optics Instance <-> Device 1 (EtherCAT)/Term 1 (EK1200)/E5 (EK1122)/X1 SP1K1-MONO(EK1100)/g_pi_up_dwn_e
//     DaqTask Inputs/PRG_DAQ_ENCODER.nEncoderCount <-> FB Inputs Channel 1/Position
//     PlcTask Inputs/Main.M7.nRawEncoderULINT <-> FB Inputs Channel 1/Position
//     PlcTask Inputs/PRG_SP1K1_MONO.gpi_upe/Count <-> FB Inputs Channel 1/Position
//   rixs_optics Instance <-> Device 1 (EtherCAT)/Term 1 (EK1200)/E5 (EK1122)/X1 SP1K1-MONO(EK1100)/m_h_e-g_h_e
//     PlcTask Inputs/Main.M8.nRawEncoderULINT <-> FB Inputs Channel 1/Position
//     PlcTask Inputs/Main.M9.nRawEncoderULINT <-> FB Inputs Channel 2/Position
//   rixs_optics Instance <-> Device 1 (EtherCAT)/Term 1 (EK1200)/E5 (EK1122)/X1 SP1K1-MONO(EK1100)/m_h_m
//     PlcTask Inputs/Main.M8.bLimitBackwardEnable <-> STM Status/Status/Digital input 2
//     PlcTask Inputs/Main.M8.bLimitForwardEnable <-> STM Status/Status/Digital input 1
//   rixs_optics Instance <-> Device 1 (EtherCAT)/Term 1 (EK1200)/E5 (EK1122)/X1 SP1K1-MONO(EK1100)/m_pi_m
//     PlcTask Inputs/Main.M6.bLimitBackwardEnable <-> STM Status/Status/Digital input 2
//     PlcTask Inputs/Main.M6.bLimitForwardEnable <-> STM Status/Status/Digital input 1
//   rixs_optics Instance <-> Device 1 (EtherCAT)/Term 1 (EK1200)/E5 (EK1122)/X1 SP1K1-MONO(EK1100)/m_pi_up_dwn_e
//     PlcTask Inputs/Main.M6.nRawEncoderULINT <-> FB Inputs Channel 2/Position
//     PlcTask Inputs/PRG_SP1K1_MONO.mpi_upe/Count <-> FB Inputs Channel 1/Position
//   rixs_optics Instance <-> Device 1 (EtherCAT)/Term 1 (EK1200)/E5 (EK1122)/X1 SP1K1-MONO(EK1100)/s_io_m
//     PlcTask Inputs/Main.M10.bLimitBackwardEnable <-> STM Status/Status/Digital input 2
//     PlcTask Inputs/Main.M10.bLimitForwardEnable <-> STM Status/Status/Digital input 1
//     PlcTask Inputs/Main.sio_current <-> STM Synchron info data/Info data 1
//     PlcTask Inputs/Main.sio_load <-> STM Synchron info data/Info data 2
//   rixs_optics Instance <-> Device 1 (EtherCAT)/Term 1 (EK1200)/EVR
//     DaqTask Inputs/PRG_DAQ_ENCODER.iLatchNeg <-> Latch/LatchNeg1
//     DaqTask Inputs/PRG_DAQ_ENCODER.iLatchPos <-> Latch/LatchPos1
//   rixs_optics Instance <-> Device 1 (EtherCAT)/Term 1 (EK1200)/PMPS_FFO
//     PlcTask Outputs/GVL_PMPS.fbFastFaultOutput1.q_xFastFaultOut <-> Channel 1/Output
//     PlcTask Outputs/GVL_PMPS.fbFastFaultOutput2.q_xFastFaultOut <-> Channel 2/Output
//   rixs_optics Instance <-> Device 1 (EtherCAT)/Term 1 (EK1200)/PMPS_PRE
//     PlcTask Inputs/PRG_2_PMPS_POST.fbArbiterIO.i_stCurrentBP <-> IO Inputs/CurrentBP
//     PlcTask Inputs/PRG_2_PMPS_POST.fbArbiterIO.xTxPDO_state <-> SYNC Inputs/TxPDO state
//     PlcTask Inputs/PRG_2_PMPS_POST.fbArbiterIO.xTxPDO_toggle <-> SYNC Inputs/TxPDO toggle
//     PlcTask Outputs/PRG_2_PMPS_POST.fbArbiterIO.q_stRequestedBP <-> IO Outputs/RequestedBP
//     PlcTask Outputs/PRG_MR1K1_BEND.nMR1K1_Y_ENC_PMPS <-> IO Outputs/MR1K1_Y_ENC
//   rixs_optics Instance <-> Device 1 (EtherCAT)/Term 1 (EK1200)/Term 5 (EK1122)/EK1100_M1K2/EL1004_M1K2_STO
//     PlcTask Inputs/PRG_MR1K2_SWITCH.M1K2.fbRunHOMS.bSTOEnable1 <-> Channel 1/Input
//     PlcTask Inputs/PRG_MR1K2_SWITCH.M1K2.fbRunHOMS.bSTOEnable2 <-> Channel 2/Input
//   rixs_optics Instance <-> Device 1 (EtherCAT)/Term 1 (EK1200)/Term 5 (EK1122)/EK1100_M1K2/EL3054_M1K2_FWM_PRSM
//     PlcTask Inputs/PRG_MR1K2_SWITCH.fM1K2_Flow_1.iRaw <-> AI Standard Channel 1/Value
//     PlcTask Inputs/PRG_MR1K2_SWITCH.fM1K2_Flow_2.iRaw <-> AI Standard Channel 2/Value
//     PlcTask Inputs/PRG_MR1K2_SWITCH.fM1K2_Press_1.iRaw <-> AI Standard Channel 3/Value
//   rixs_optics Instance <-> Device 1 (EtherCAT)/Term 1 (EK1200)/Term 5 (EK1122)/EK1100_M1K2/EL5042_M1K2_Pitch
//     PlcTask Inputs/GVL_M1K1.M1K1_Pitch.diEncCnt <-> FB Inputs Channel 1/Position
//     PlcTask Inputs/GVL_M1K2.M1K2_Pitch.diEncCnt <-> FB Inputs Channel 1/Position
//     PlcTask Inputs/Main.M5.nRawEncoderULINT <-> FB Inputs Channel 1/Position
//   rixs_optics Instance <-> Device 1 (EtherCAT)/Term 1 (EK1200)/Term 5 (EK1122)/EK1100_M1K2/EL5042_M1K2_Xupdwn
//     PlcTask Inputs/Main.M3.nRawEncoderULINT <-> FB Inputs Channel 1/Position
//     PlcTask Inputs/Main.M4.nRawEncoderULINT <-> FB Inputs Channel 1/Position
//     PlcTask Inputs/PRG_MR1K2_SWITCH.M1K2.fbRunHOMS.stXdwnEnc/Count <-> FB Inputs Channel 2/Position
//     PlcTask Inputs/PRG_MR1K2_SWITCH.M1K2.fbRunHOMS.stXupEnc/Count <-> FB Inputs Channel 1/Position
//   rixs_optics Instance <-> Device 1 (EtherCAT)/Term 1 (EK1200)/Term 5 (EK1122)/EK1100_M1K2/EL5042_M1K2_Yleftright
//     PlcTask Inputs/Main.M1.nRawEncoderULINT <-> FB Inputs Channel 1/Position
//     PlcTask Inputs/Main.M2.nRawEncoderULINT <-> FB Inputs Channel 2/Position
//     PlcTask Inputs/PRG_MR1K2_SWITCH.M1K2.fbRunHOMS.stYdwnEnc/Count <-> FB Inputs Channel 2/Position
//     PlcTask Inputs/PRG_MR1K2_SWITCH.M1K2.fbRunHOMS.stYupEnc/Count <-> FB Inputs Channel 1/Position
//   rixs_optics Instance <-> Device 1 (EtherCAT)/Term 1 (EK1200)/Term 5 (EK1122)/EK1100_M1K2/EL6001_M1K2_PitchFine
//     SerialIO Inputs/GVL_SerialIO.Serial_stComIn_M1K2/D[{0..21}] <-> COM Inputs/Data In {0..21}  (22 links)
//     SerialIO Inputs/GVL_SerialIO.Serial_stComIn_M1K2/Status <-> COM Inputs/Status
//     SerialIO Outputs/GVL_SerialIO.Serial_stComOut_M1K2/Ctrl <-> COM Outputs/Ctrl
//     SerialIO Outputs/GVL_SerialIO.Serial_stComOut_M1K2/D[{0..21}] <-> COM Outputs/Data Out {0..21}  (22 links)
//   rixs_optics Instance <-> Device 1 (EtherCAT)/Term 1 (EK1200)/Term 5 (EK1122)/EK1100_M1K2/EL7047_M1K2_PitchCoarse
//     PlcTask Inputs/Main.M5.bLimitBackwardEnable <-> STM Status/Status/Digital input 2
//     PlcTask Inputs/Main.M5.bLimitForwardEnable <-> STM Status/Status/Digital input 1
//   rixs_optics Instance <-> Device 1 (EtherCAT)/Term 1 (EK1200)/Term 5 (EK1122)/EK1100_M1K2/EL7047_M1K2_Xdwn
//     PlcTask Inputs/Main.M4.bLimitBackwardEnable <-> STM Status/Status/Digital input 2
//     PlcTask Inputs/Main.M4.bLimitForwardEnable <-> STM Status/Status/Digital input 1
//     PlcTask Inputs/PRG_MR1K2_SWITCH.M1K2.fMotorCurSecondX <-> STM Synchron info data/Info data 2
//     PlcTask Inputs/PRG_MR1K2_SWITCH.M1K2.fSupplySecondX <-> STM Synchron info data/Info data 1
//   rixs_optics Instance <-> Device 1 (EtherCAT)/Term 1 (EK1200)/Term 5 (EK1122)/EK1100_M1K2/EL7047_M1K2_Xup
//     PlcTask Inputs/Main.M3.bLimitBackwardEnable <-> STM Status/Status/Digital input 2
//     PlcTask Inputs/Main.M3.bLimitForwardEnable <-> STM Status/Status/Digital input 1
//   rixs_optics Instance <-> Device 1 (EtherCAT)/Term 1 (EK1200)/Term 5 (EK1122)/EK1100_M1K2/EL7047_M1K2_Yleft
//     PlcTask Inputs/Main.M1.bLimitBackwardEnable <-> STM Status/Status/Digital input 2
//     PlcTask Inputs/Main.M1.bLimitForwardEnable <-> STM Status/Status/Digital input 1
//   rixs_optics Instance <-> Device 1 (EtherCAT)/Term 1 (EK1200)/Term 5 (EK1122)/EK1100_M1K2/EL7047_M1K2_Yright
//     PlcTask Inputs/Main.M2.bLimitBackwardEnable <-> STM Status/Status/Digital input 2
//     PlcTask Inputs/Main.M2.bLimitForwardEnable <-> STM Status/Status/Digital input 1
//     PlcTask Inputs/PRG_MR1K2_SWITCH.M1K2.fMotorCurSecondY <-> STM Synchron info data/Info data 2
//     PlcTask Inputs/PRG_MR1K2_SWITCH.M1K2.fSupplySecondY <-> STM Synchron info data/Info data 1
//   rixs_optics Instance <-> Device 1 (EtherCAT)/Term 1 (EK1200)/Term 5 (EK1122)/EK1100_MR1K1/EL1004_M1K1_STO
//     PlcTask Inputs/PRG_MR1K1_BEND.M1K1.fbRunHOMS.bSTOEnable1 <-> Channel 1/Input
//     PlcTask Inputs/PRG_MR1K1_BEND.M1K1.fbRunHOMS.bSTOEnable2 <-> Channel 2/Input
//   rixs_optics Instance <-> Device 1 (EtherCAT)/Term 1 (EK1200)/Term 5 (EK1122)/EK1100_MR1K1/EL3054_M1K1_FWM_PRSM
//     PlcTask Inputs/PRG_MR1K1_BEND.fM1K1_Flow_1.iRaw <-> AI Standard Channel 1/Value
//     PlcTask Inputs/PRG_MR1K1_BEND.fM1K1_Flow_2.iRaw <-> AI Standard Channel 2/Value
//     PlcTask Inputs/PRG_MR1K1_BEND.fM1K1_Press_1.iRaw <-> AI Standard Channel 3/Value
//   rixs_optics Instance <-> Device 1 (EtherCAT)/Term 1 (EK1200)/Term 5 (EK1122)/EK1100_MR1K1/EL3202-0010-XUP-XDWN
//     PlcTask Inputs/PRG_MR1K1_BEND.fbXDWNMotorTemp.iRaw <-> RTD Inputs Channel 2/Value
//     PlcTask Inputs/PRG_MR1K1_BEND.fbXUPMotorTemp.iRaw <-> RTD Inputs Channel 1/Value
//   rixs_optics Instance <-> Device 1 (EtherCAT)/Term 1 (EK1200)/Term 5 (EK1122)/EK1100_MR1K1/EL3202-0010-YUP-YDWN
//     PlcTask Inputs/PRG_MR1K1_BEND.fbYDWNMotorTemp.iRaw <-> RTD Inputs Channel 2/Value
//     PlcTask Inputs/PRG_MR1K1_BEND.fbYUPMotorTemp.iRaw <-> RTD Inputs Channel 1/Value
//   rixs_optics Instance <-> Device 1 (EtherCAT)/Term 1 (EK1200)/Term 5 (EK1122)/EK1100_MR1K1/EL5042_M1K1_Pitch
//     PlcTask Inputs/Main.M16.nRawEncoderULINT <-> FB Inputs Channel 1/Position
//   rixs_optics Instance <-> Device 1 (EtherCAT)/Term 1 (EK1200)/Term 5 (EK1122)/EK1100_MR1K1/EL5042_M1K1_Xupdwn
//     PlcTask Inputs/Main.M14.nRawEncoderULINT <-> FB Inputs Channel 1/Position
//     PlcTask Inputs/PRG_MR1K1_BEND.M1K1.fbRunHOMS.stXdwnEnc/Count <-> FB Inputs Channel 2/Position
//     PlcTask Inputs/PRG_MR1K1_BEND.M1K1.fbRunHOMS.stXupEnc/Count <-> FB Inputs Channel 1/Position
//   rixs_optics Instance <-> Device 1 (EtherCAT)/Term 1 (EK1200)/Term 5 (EK1122)/EK1100_MR1K1/EL5042_M1K1_Yupdwn
//     PlcTask Inputs/Main.M12.nRawEncoderULINT <-> FB Inputs Channel 1/Position
//     PlcTask Inputs/PRG_MR1K1_BEND.M1K1.fbRunHOMS.stYdwnEnc/Count <-> FB Inputs Channel 2/Position
//     PlcTask Inputs/PRG_MR1K1_BEND.M1K1.fbRunHOMS.stYupEnc/Count <-> FB Inputs Channel 1/Position
//     PlcTask Inputs/PRG_MR1K1_BEND.bMR1K1_Y_ENC_Ready <-> FB Inputs Channel 1/Status/Ready
//     PlcTask Inputs/PRG_MR1K1_BEND.bMR1K1_Y_ENC_TxPDO <-> FB Inputs Channel 1/Status/TxPDO State
//   rixs_optics Instance <-> Device 1 (EtherCAT)/Term 1 (EK1200)/Term 5 (EK1122)/EK1100_MR1K1/EL7047_M1K1_PitchCoarse
//     PlcTask Inputs/Main.M16.bLimitBackwardEnable <-> STM Status/Status/Digital input 2
//     PlcTask Inputs/Main.M16.bLimitForwardEnable <-> STM Status/Status/Digital input 1
//   rixs_optics Instance <-> Device 1 (EtherCAT)/Term 1 (EK1200)/Term 5 (EK1122)/EK1100_MR1K1/EL7047_M1K1_Xdwn
//     PlcTask Inputs/Main.M15.bLimitBackwardEnable <-> STM Status/Status/Digital input 2
//     PlcTask Inputs/Main.M15.bLimitForwardEnable <-> STM Status/Status/Digital input 1
//     PlcTask Inputs/PRG_MR1K1_BEND.M1K1.fMotorCurSecondX <-> STM Synchron info data/Info data 2
//     PlcTask Inputs/PRG_MR1K1_BEND.M1K1.fSupplySecondX <-> STM Synchron info data/Info data 1
//   rixs_optics Instance <-> Device 1 (EtherCAT)/Term 1 (EK1200)/Term 5 (EK1122)/EK1100_MR1K1/EL7047_M1K1_Xup
//     PlcTask Inputs/Main.M14.bLimitBackwardEnable <-> STM Status/Status/Digital input 2
//     PlcTask Inputs/Main.M14.bLimitForwardEnable <-> STM Status/Status/Digital input 1
//   rixs_optics Instance <-> Device 1 (EtherCAT)/Term 1 (EK1200)/Term 5 (EK1122)/EK1100_MR1K1/EL7047_M1K1_Ydwn
//     PlcTask Inputs/Main.M12.bLimitBackwardEnable <-> STM Status/Status/Digital input 2
//     PlcTask Inputs/Main.M13.bLimitBackwardEnable <-> STM Status/Status/Digital input 2
//     PlcTask Inputs/Main.M12.bLimitForwardEnable <-> STM Status/Status/Digital input 1
//     PlcTask Inputs/Main.M13.bLimitForwardEnable <-> STM Status/Status/Digital input 1
//     PlcTask Inputs/PRG_MR1K1_BEND.M1K1.fMotorCurSecondY <-> STM Synchron info data/Info data 2
//     PlcTask Inputs/PRG_MR1K1_BEND.M1K1.fSupplySecondY <-> STM Synchron info data/Info data 1
//   rixs_optics Instance <-> Device 1 (EtherCAT)/Term 1 (EK1200)/Term 5 (EK1122)/EK1100_MR1K1_BEND/EL1004_M1K1_BENDER_STO
//     PlcTask Inputs/PRG_MR1K1_BEND_BENDER.M1K1BENDbSTOEnable1 <-> Channel 1/Input
//     PlcTask Inputs/PRG_MR1K1_BEND_BENDER.M1K1BENDbSTOEnable2 <-> Channel 2/Input
//   rixs_optics Instance <-> Device 1 (EtherCAT)/Term 1 (EK1200)/Term 5 (EK1122)/EK1100_MR1K1_BEND/EL2024-0010_M1K1_BEND_LED1
//     PlcTask Outputs/PRG_MR1K1_BEND.bLEDPower01 <-> Channel 1/Output
//     PlcTask Outputs/PRG_MR1K1_BEND.bLEDPower02 <-> Channel 2/Output
//     PlcTask Outputs/PRG_MR1K1_BEND.bLEDPower03 <-> Channel 3/Output
//     PlcTask Outputs/PRG_MR1K1_BEND.bLEDPower04 <-> Channel 4/Output
//   rixs_optics Instance <-> Device 1 (EtherCAT)/Term 1 (EK1200)/Term 5 (EK1122)/EK1100_MR1K1_BEND/EL3202-0010_M1K1DS2_M1K1DS3
//     PlcTask Inputs/GVL_M1K1_BENDER_RTD.nM1K1DS_RTD_2 <-> RTD Inputs Channel 1/Value
//     PlcTask Inputs/GVL_M1K1_BENDER_RTD.nM1K1DS_RTD_3 <-> RTD Inputs Channel 2/Value
//   rixs_optics Instance <-> Device 1 (EtherCAT)/Term 1 (EK1200)/Term 5 (EK1122)/EK1100_MR1K1_BEND/EL3202-0010_M1K1US1_M1K1US2
//     PlcTask Inputs/GVL_M1K1_BENDER_RTD.nM1K1US_RTD_1 <-> RTD Inputs Channel 1/Value
//     PlcTask Inputs/GVL_M1K1_BENDER_RTD.nM1K1US_RTD_2 <-> RTD Inputs Channel 2/Value
//   rixs_optics Instance <-> Device 1 (EtherCAT)/Term 1 (EK1200)/Term 5 (EK1122)/EK1100_MR1K1_BEND/EL3202-0010_M1K1US3_M1K1DS1
//     PlcTask Inputs/GVL_M1K1_BENDER_RTD.nM1K1DS_RTD_1 <-> RTD Inputs Channel 2/Value
//     PlcTask Inputs/GVL_M1K1_BENDER_RTD.nM1K1US_RTD_3 <-> RTD Inputs Channel 1/Value
//   rixs_optics Instance <-> Device 1 (EtherCAT)/Term 1 (EK1200)/Term 5 (EK1122)/EK1100_MR1K1_BEND/EL5042_M1K1_BEND_USDS
//     PlcTask Inputs/Main.M17.nRawEncoderULINT <-> FB Inputs Channel 1/Position
//     PlcTask Inputs/Main.M18.nRawEncoderULINT <-> FB Inputs Channel 2/Position
//   rixs_optics Instance <-> Device 1 (EtherCAT)/Term 1 (EK1200)/Term 5 (EK1122)/EK1100_MR1K1_BEND/EL7041_M1K1_BEND_DS
//     PlcTask Inputs/Main.M18.bLimitBackwardEnable <-> STM Status/Status/Digital input 2
//     PlcTask Inputs/Main.M18.bLimitForwardEnable <-> STM Status/Status/Digital input 1
//   rixs_optics Instance <-> Device 1 (EtherCAT)/Term 1 (EK1200)/Term 5 (EK1122)/EK1100_MR1K1_BEND/EL7041_M1K1_BEND_US
//     PlcTask Inputs/Main.M17.bLimitBackwardEnable <-> STM Status/Status/Digital input 2
//   rixs_optics Instance <-> Device 1 (EtherCAT)/Term 1 (EK1200)/Term 5 (EK1122)/EK1100_ST1K2_ZOS/ST1K1-EL2008
//     PlcTask Outputs/Main.M24.bBrakeRelease <-> Channel 1/Output
//   rixs_optics Instance <-> Device 1 (EtherCAT)/Term 1 (EK1200)/Term 5 (EK1122)/EK1100_ST1K2_ZOS/ST1K1-EL5042
//     PlcTask Inputs/Main.M24.nRawEncoderULINT <-> FB Inputs Channel 1/Position
//   rixs_optics Instance <-> Device 1 (EtherCAT)/Term 1 (EK1200)/Term 5 (EK1122)/EK1100_ST1K2_ZOS/ST1K1-EL7041
//     PlcTask Inputs/Main.M24.bLimitBackwardEnable <-> STM Status/Status/Digital input 2
//     PlcTask Inputs/Main.M24.bLimitForwardEnable <-> STM Status/Status/Digital input 1
//   rixs_optics Instance <-> Device 1 (EtherCAT)/Term 1 (EK1200)/Term 79 (EK1521-0010)/Term 306 (EK1501-0010)/Term 310 (EK1122)/EK1100_MR2K2/EL1004_M2K2_STO
//     PlcTask Inputs/PRG_MR2K2_FLAT.M2K2FLATbSTOEnable1 <-> Channel 1/Input
//     PlcTask Inputs/PRG_MR2K2_FLAT.M2K2FLATbSTOEnable2 <-> Channel 2/Input
//   rixs_optics Instance <-> Device 1 (EtherCAT)/Term 1 (EK1200)/Term 79 (EK1521-0010)/Term 306 (EK1501-0010)/Term 310 (EK1122)/EK1100_MR2K2/EL3054_MR2K2_FWM_PRSM
//     PlcTask Inputs/PRG_MR2K2_FLAT.fbCoolingPanel.fbFlow_1.iRaw <-> AI Standard Channel 1/Value
//     PlcTask Inputs/PRG_MR2K2_FLAT.fbCoolingPanel.fbFlow_2.iRaw <-> AI Standard Channel 3/Value
//     PlcTask Inputs/PRG_MR2K2_FLAT.fbCoolingPanel.fbPress_1.iRaw <-> AI Standard Channel 2/Value
//   rixs_optics Instance <-> Device 1 (EtherCAT)/Term 1 (EK1200)/Term 79 (EK1521-0010)/Term 306 (EK1501-0010)/Term 310 (EK1122)/EK1100_MR2K2/EL5042_M2K2X_M2K2Y
//     PlcTask Inputs/Main.M25.nRawEncoderULINT <-> FB Inputs Channel 1/Position
//     PlcTask Inputs/Main.M26.nRawEncoderULINT <-> FB Inputs Channel 2/Position
//   rixs_optics Instance <-> Device 1 (EtherCAT)/Term 1 (EK1200)/Term 79 (EK1521-0010)/Term 306 (EK1501-0010)/Term 310 (EK1122)/EK1100_MR2K2/EL5042_M2K2rX
//     PlcTask Inputs/Main.M27.nRawEncoderULINT <-> FB Inputs Channel 1/Position
//   rixs_optics Instance <-> Device 1 (EtherCAT)/Term 1 (EK1200)/Term 79 (EK1521-0010)/Term 306 (EK1501-0010)/Term 310 (EK1122)/EK1100_MR2K2/EL7041_M2K2X
//     PlcTask Inputs/Main.M25.bLimitBackwardEnable <-> STM Status/Status/Digital input 2
//     PlcTask Inputs/Main.M25.bLimitForwardEnable <-> STM Status/Status/Digital input 1
//   rixs_optics Instance <-> Device 1 (EtherCAT)/Term 1 (EK1200)/Term 79 (EK1521-0010)/Term 306 (EK1501-0010)/Term 310 (EK1122)/EK1100_MR2K2/EL7041_M2K2Y
//     PlcTask Inputs/Main.M26.bLimitBackwardEnable <-> STM Status/Status/Digital input 2
//     PlcTask Inputs/Main.M26.bLimitForwardEnable <-> STM Status/Status/Digital input 1
//   rixs_optics Instance <-> Device 1 (EtherCAT)/Term 1 (EK1200)/Term 79 (EK1521-0010)/Term 306 (EK1501-0010)/Term 310 (EK1122)/EK1100_MR2K2/EL7041_M2K2rX
//     PlcTask Inputs/Main.M27.bLimitBackwardEnable <-> STM Status/Status/Digital input 1
//     PlcTask Inputs/Main.M27.bLimitForwardEnable <-> STM Status/Status/Digital input 2
//   rixs_optics Instance <-> Device 1 (EtherCAT)/Term 1 (EK1200)/Term 79 (EK1521-0010)/Term 306 (EK1501-0010)/Term 310 (EK1122)/EK1100_MR3K2/EL5042_M3K2X_M3K2Y
//     PlcTask Inputs/Main.M28.nRawEncoderULINT <-> FB Inputs Channel 1/Position
//     PlcTask Inputs/Main.M29.nRawEncoderULINT <-> FB Inputs Channel 2/Position
//   rixs_optics Instance <-> Device 1 (EtherCAT)/Term 1 (EK1200)/Term 79 (EK1521-0010)/Term 306 (EK1501-0010)/Term 310 (EK1122)/EK1100_MR3K2/EL5042_M3K2rY
//     PlcTask Inputs/Main.M30.nRawEncoderULINT <-> FB Inputs Channel 1/Position
//   rixs_optics Instance <-> Device 1 (EtherCAT)/Term 1 (EK1200)/Term 79 (EK1521-0010)/Term 306 (EK1501-0010)/Term 310 (EK1122)/EK1100_MR3K2/EL7041_M3K2X
//     PlcTask Inputs/Main.M28.bLimitBackwardEnable <-> STM Status/Status/Digital input 2
//     PlcTask Inputs/Main.M28.bLimitForwardEnable <-> STM Status/Status/Digital input 1
//   rixs_optics Instance <-> Device 1 (EtherCAT)/Term 1 (EK1200)/Term 79 (EK1521-0010)/Term 306 (EK1501-0010)/Term 310 (EK1122)/EK1100_MR3K2/EL7041_M3K2Y
//     PlcTask Inputs/Main.M29.bLimitBackwardEnable <-> STM Status/Status/Digital input 2
//     PlcTask Inputs/Main.M29.bLimitForwardEnable <-> STM Status/Status/Digital input 1
//   rixs_optics Instance <-> Device 1 (EtherCAT)/Term 1 (EK1200)/Term 79 (EK1521-0010)/Term 306 (EK1501-0010)/Term 310 (EK1122)/EK1100_MR3K2/EL7041_M3K2rY
//     PlcTask Inputs/Main.M30.bLimitBackwardEnable <-> STM Status/Status/Digital input 2
//     PlcTask Inputs/Main.M30.bLimitForwardEnable <-> STM Status/Status/Digital input 1
//   rixs_optics Instance <-> Device 1 (EtherCAT)/Term 1 (EK1200)/Term 79 (EK1521-0010)/Term 306 (EK1501-0010)/Term 310 (EK1122)/EK1100_MR3K2_BENDER/EL1004_M3K2_STO
//     PlcTask Inputs/PRG_MR3K2_KBH.M3K2KBHbSTOEnable1 <-> Channel 1/Input
//     PlcTask Inputs/PRG_MR3K2_KBH.M3K2KBHbSTOEnable2 <-> Channel 2/Input
//   rixs_optics Instance <-> Device 1 (EtherCAT)/Term 1 (EK1200)/Term 79 (EK1521-0010)/Term 306 (EK1501-0010)/Term 310 (EK1122)/EK1100_MR3K2_BENDER/EL3202-0010_M3K2DS2_M3K2DS3
//     PlcTask Inputs/GVL_M3K2.nM3K2DS_RTD_3 <-> RTD Inputs Channel 2/Value
//     PlcTask Inputs/PRG_MR3K2_KBH.fbM3K2_Chin_Right_RTD.bError <-> RTD Inputs Channel 1/Status/Error
//     PlcTask Inputs/PRG_MR3K2_KBH.fbM3K2_Chin_Right_RTD.bOverrange <-> RTD Inputs Channel 1/Status/Overrange
//     PlcTask Inputs/PRG_MR3K2_KBH.fbM3K2_Chin_Right_RTD.bUnderrange <-> RTD Inputs Channel 1/Status/Underrange
//     PlcTask Inputs/PRG_MR3K2_KBH.fbM3K2_Chin_Right_RTD.iRaw <-> RTD Inputs Channel 1/Value
//   rixs_optics Instance <-> Device 1 (EtherCAT)/Term 1 (EK1200)/Term 79 (EK1521-0010)/Term 306 (EK1501-0010)/Term 310 (EK1122)/EK1100_MR3K2_BENDER/EL3202-0010_M3K2US1_M3K2US2
//     PlcTask Inputs/GVL_M3K2.nM3K2US_RTD_1 <-> RTD Inputs Channel 1/Value
//     PlcTask Inputs/GVL_M3K2.nM3K2US_RTD_2 <-> RTD Inputs Channel 2/Value
//   rixs_optics Instance <-> Device 1 (EtherCAT)/Term 1 (EK1200)/Term 79 (EK1521-0010)/Term 306 (EK1501-0010)/Term 310 (EK1122)/EK1100_MR3K2_BENDER/EL3202-0010_M3K2US3_M3K2DS1
//     PlcTask Inputs/GVL_M3K2.nM3K2DS_RTD_1 <-> RTD Inputs Channel 2/Value
//     PlcTask Inputs/PRG_MR3K2_KBH.fbM3K2_Chin_Left_RTD.bError <-> RTD Inputs Channel 1/Status/Error
//     PlcTask Inputs/PRG_MR3K2_KBH.fbM3K2_Chin_Left_RTD.bOverrange <-> RTD Inputs Channel 1/Status/Overrange
//     PlcTask Inputs/PRG_MR3K2_KBH.fbM3K2_Chin_Left_RTD.bUnderrange <-> RTD Inputs Channel 1/Status/Underrange
//     PlcTask Inputs/PRG_MR3K2_KBH.fbM3K2_Chin_Left_RTD.iRaw <-> RTD Inputs Channel 1/Value
//   rixs_optics Instance <-> Device 1 (EtherCAT)/Term 1 (EK1200)/Term 79 (EK1521-0010)/Term 306 (EK1501-0010)/Term 310 (EK1122)/EK1100_MR3K2_BENDER/EL5042_M3K2_BEND_USDS
//     PlcTask Inputs/Main.M31.nRawEncoderULINT <-> FB Inputs Channel 1/Position
//     PlcTask Inputs/Main.M32.nRawEncoderULINT <-> FB Inputs Channel 2/Position
//   rixs_optics Instance <-> Device 1 (EtherCAT)/Term 1 (EK1200)/Term 79 (EK1521-0010)/Term 306 (EK1501-0010)/Term 310 (EK1122)/EK1100_MR3K2_BENDER/EL7041_M3K2_BEND_DS
//     PlcTask Inputs/Main.M32.bLimitBackwardEnable <-> STM Status/Status/Digital input 2
//     PlcTask Inputs/Main.M32.bLimitForwardEnable <-> STM Status/Status/Digital input 1
//   rixs_optics Instance <-> Device 1 (EtherCAT)/Term 1 (EK1200)/Term 79 (EK1521-0010)/Term 306 (EK1501-0010)/Term 310 (EK1122)/EK1100_MR3K2_BENDER/EL7041_M3K2_BEND_US
//     PlcTask Inputs/Main.M31.bLimitBackwardEnable <-> STM Status/Status/Digital input 2
//     PlcTask Inputs/Main.M31.bLimitForwardEnable <-> STM Status/Status/Digital input 1
//   rixs_optics Instance <-> Device 1 (EtherCAT)/Term 1 (EK1200)/Term 79 (EK1521-0010)/Term 306 (EK1501-0010)/Term 322 (EK1122)/EK1100_MR4K2/EL3054_MR3_4K2_FWM_PRSM
//     PlcTask Inputs/PRG_MR3K2_KBH.fbCoolingPanel.fbFlow_1.iRaw <-> AI Standard Channel 1/Value
//     PlcTask Inputs/PRG_MR3K2_KBH.fbCoolingPanel.fbPress_1.iRaw <-> AI Standard Channel 2/Value
//     PlcTask Inputs/PRG_MR4K2_KBV.fbCoolingPanel.fbFlow_1.iRaw <-> AI Standard Channel 3/Value
//     PlcTask Inputs/PRG_MR4K2_KBV.fbCoolingPanel.fbPress_1.iRaw <-> AI Standard Channel 2/Value
//   rixs_optics Instance <-> Device 1 (EtherCAT)/Term 1 (EK1200)/Term 79 (EK1521-0010)/Term 306 (EK1501-0010)/Term 322 (EK1122)/EK1100_MR4K2/EL5042_M4K2X_M4K2Y
//     PlcTask Inputs/Main.M33.nRawEncoderULINT <-> FB Inputs Channel 1/Position
//     PlcTask Inputs/Main.M34.nRawEncoderULINT <-> FB Inputs Channel 2/Position
//   rixs_optics Instance <-> Device 1 (EtherCAT)/Term 1 (EK1200)/Term 79 (EK1521-0010)/Term 306 (EK1501-0010)/Term 322 (EK1122)/EK1100_MR4K2/EL5042_M4K2rX
//     PlcTask Inputs/Main.M35.nRawEncoderULINT <-> FB Inputs Channel 1/Position
//   rixs_optics Instance <-> Device 1 (EtherCAT)/Term 1 (EK1200)/Term 79 (EK1521-0010)/Term 306 (EK1501-0010)/Term 322 (EK1122)/EK1100_MR4K2/EL7041_M4K2X
//     PlcTask Inputs/Main.M33.bLimitBackwardEnable <-> STM Status/Status/Digital input 2
//     PlcTask Inputs/Main.M33.bLimitForwardEnable <-> STM Status/Status/Digital input 1
//   rixs_optics Instance <-> Device 1 (EtherCAT)/Term 1 (EK1200)/Term 79 (EK1521-0010)/Term 306 (EK1501-0010)/Term 322 (EK1122)/EK1100_MR4K2/EL7041_M4K2Y
//     PlcTask Inputs/Main.M34.bLimitBackwardEnable <-> STM Status/Status/Digital input 2
//     PlcTask Inputs/Main.M34.bLimitForwardEnable <-> STM Status/Status/Digital input 1
//   rixs_optics Instance <-> Device 1 (EtherCAT)/Term 1 (EK1200)/Term 79 (EK1521-0010)/Term 306 (EK1501-0010)/Term 322 (EK1122)/EK1100_MR4K2/EL7041_M4K2rX
//     PlcTask Inputs/Main.M35.bLimitBackwardEnable <-> STM Status/Status/Digital input 2
//     PlcTask Inputs/Main.M35.bLimitForwardEnable <-> STM Status/Status/Digital input 1
//   rixs_optics Instance <-> Device 1 (EtherCAT)/Term 1 (EK1200)/Term 79 (EK1521-0010)/Term 306 (EK1501-0010)/Term 322 (EK1122)/EK1100_MR4K2_BENDER/EL1004_M4K2_STO
//     PlcTask Inputs/PRG_MR4K2_KBV.M4K2KBVbSTOEnable1 <-> Channel 1/Input
//     PlcTask Inputs/PRG_MR4K2_KBV.M4K2KBVbSTOEnable2 <-> Channel 2/Input
//   rixs_optics Instance <-> Device 1 (EtherCAT)/Term 1 (EK1200)/Term 79 (EK1521-0010)/Term 306 (EK1501-0010)/Term 322 (EK1122)/EK1100_MR4K2_BENDER/EL3202-0010_M4K2US1_M4K2US2
//     PlcTask Inputs/GVL_M4K2.nM4K2US_RTD_1 <-> RTD Inputs Channel 1/Value
//     PlcTask Inputs/GVL_M4K2.nM4K2US_RTD_2 <-> RTD Inputs Channel 2/Value
//   rixs_optics Instance <-> Device 1 (EtherCAT)/Term 1 (EK1200)/Term 79 (EK1521-0010)/Term 306 (EK1501-0010)/Term 322 (EK1122)/EK1100_MR4K2_BENDER/EL3202-0010_M4K2US3_M4K2DS1
//     PlcTask Inputs/GVL_M4K2.nM4K2DS_RTD_1 <-> RTD Inputs Channel 2/Value
//     PlcTask Inputs/GVL_M4K2.nM4K2US_RTD_3 <-> RTD Inputs Channel 1/Value
//   rixs_optics Instance <-> Device 1 (EtherCAT)/Term 1 (EK1200)/Term 79 (EK1521-0010)/Term 306 (EK1501-0010)/Term 322 (EK1122)/EK1100_MR4K2_BENDER/EL3204_M4K2_CHIN
//     PlcTask Inputs/PRG_MR4K2_KBV.fbM4K2_Chin_Left_RTD.bError <-> RTD Inputs Channel 2/Status/Error
//     PlcTask Inputs/PRG_MR4K2_KBV.fbM4K2_Chin_Left_RTD.bOverrange <-> RTD Inputs Channel 2/Status/Overrange
//     PlcTask Inputs/PRG_MR4K2_KBV.fbM4K2_Chin_Left_RTD.bUnderrange <-> RTD Inputs Channel 2/Status/Underrange
//     PlcTask Inputs/PRG_MR4K2_KBV.fbM4K2_Chin_Left_RTD.iRaw <-> RTD Inputs Channel 2/Value
//     PlcTask Inputs/PRG_MR4K2_KBV.fbM4K2_Chin_Right_RTD.bError <-> RTD Inputs Channel 1/Status/Error
//     PlcTask Inputs/PRG_MR4K2_KBV.fbM4K2_Chin_Right_RTD.bOverrange <-> RTD Inputs Channel 1/Status/Overrange
//     PlcTask Inputs/PRG_MR4K2_KBV.fbM4K2_Chin_Right_RTD.bUnderrange <-> RTD Inputs Channel 1/Status/Underrange
//     PlcTask Inputs/PRG_MR4K2_KBV.fbM4K2_Chin_Right_RTD.iRaw <-> RTD Inputs Channel 1/Value
//   rixs_optics Instance <-> Device 1 (EtherCAT)/Term 1 (EK1200)/Term 79 (EK1521-0010)/Term 306 (EK1501-0010)/Term 322 (EK1122)/EK1100_MR4K2_BENDER/EL5042_M4K2_BEND_USDS
//     PlcTask Inputs/Main.M36.nRawEncoderULINT <-> FB Inputs Channel 1/Position
//     PlcTask Inputs/Main.M37.nRawEncoderULINT <-> FB Inputs Channel 2/Position
//   rixs_optics Instance <-> Device 1 (EtherCAT)/Term 1 (EK1200)/Term 79 (EK1521-0010)/Term 306 (EK1501-0010)/Term 322 (EK1122)/EK1100_MR4K2_BENDER/EL7041_M4K2_BEND_DS
//     PlcTask Inputs/Main.M37.bLimitBackwardEnable <-> STM Status/Status/Digital input 2
//     PlcTask Inputs/Main.M37.bLimitForwardEnable <-> STM Status/Status/Digital input 1
//   rixs_optics Instance <-> Device 1 (EtherCAT)/Term 1 (EK1200)/Term 79 (EK1521-0010)/Term 306 (EK1501-0010)/Term 322 (EK1122)/EK1100_MR4K2_BENDER/EL7041_M4K2_BEND_US
//     PlcTask Inputs/Main.M36.bLimitBackwardEnable <-> STM Status/Status/Digital input 2
//     PlcTask Inputs/Main.M36.bLimitForwardEnable <-> STM Status/Status/Digital input 1
//   rixs_optics Instance <-> NC-Task 1 SAF/Axes/Axis 24 ST1K1-ZOS-MMS
//     PlcTask Inputs/Main.M24.Axis.NcToPlc <-> Outputs/ToPlc
//     PlcTask Outputs/Main.M24.Axis.PlcToNc <-> Inputs/FromPlc
//   rixs_optics Instance <-> NC-Task 1 SAF/Axes/M1K1-BEND-DS
//     PlcTask Inputs/Main.M18.Axis.NcToPlc <-> Outputs/ToPlc
//     PlcTask Outputs/Main.M18.Axis.PlcToNc <-> Inputs/FromPlc
//   rixs_optics Instance <-> NC-Task 1 SAF/Axes/M1K1-BEND-US
//     PlcTask Inputs/Main.M17.Axis.NcToPlc <-> Outputs/ToPlc
//     PlcTask Outputs/Main.M17.Axis.PlcToNc <-> Inputs/FromPlc
//   rixs_optics Instance <-> NC-Task 1 SAF/Axes/M1K1-Pitch
//     PlcTask Outputs/Main.M16.Axis.PlcToNc <-> Inputs/FromPlc
//     StatsTask Inputs/Main.M16.Axis.NcToPlc <-> Outputs/ToPlc
//   rixs_optics Instance <-> NC-Task 1 SAF/Axes/M1K1-Xdwn
//     PlcTask Inputs/Main.M15.Axis.NcToPlc <-> Outputs/ToPlc
//     PlcTask Outputs/Main.M15.Axis.PlcToNc <-> Inputs/FromPlc
//   rixs_optics Instance <-> NC-Task 1 SAF/Axes/M1K1-Xup
//     PlcTask Inputs/Main.M14.Axis.NcToPlc <-> Outputs/ToPlc
//     PlcTask Outputs/Main.M14.Axis.PlcToNc <-> Inputs/FromPlc
//   rixs_optics Instance <-> NC-Task 1 SAF/Axes/M1K1-Ydwn
//     PlcTask Inputs/Main.M13.Axis.NcToPlc <-> Outputs/ToPlc
//     PlcTask Outputs/Main.M13.Axis.PlcToNc <-> Inputs/FromPlc
//   rixs_optics Instance <-> NC-Task 1 SAF/Axes/M1K1-Yup
//     PlcTask Inputs/Main.M12.Axis.NcToPlc <-> Outputs/ToPlc
//     PlcTask Outputs/Main.M12.Axis.PlcToNc <-> Inputs/FromPlc
//   rixs_optics Instance <-> NC-Task 1 SAF/Axes/M1K2-Pitch
//     PlcTask Inputs/Main.M5.Axis.NcToPlc <-> Outputs/ToPlc
//     PlcTask Outputs/Main.M5.Axis.PlcToNc <-> Inputs/FromPlc
//   rixs_optics Instance <-> NC-Task 1 SAF/Axes/M1K2-Xdwn
//     PlcTask Inputs/Main.M4.Axis.NcToPlc <-> Outputs/ToPlc
//     PlcTask Outputs/Main.M4.Axis.PlcToNc <-> Inputs/FromPlc
//   rixs_optics Instance <-> NC-Task 1 SAF/Axes/M1K2-Xup
//     PlcTask Inputs/Main.M3.Axis.NcToPlc <-> Outputs/ToPlc
//     PlcTask Outputs/Main.M3.Axis.PlcToNc <-> Inputs/FromPlc
//   rixs_optics Instance <-> NC-Task 1 SAF/Axes/M1K2-Yleft
//     PlcTask Inputs/Main.M1.Axis.NcToPlc <-> Outputs/ToPlc
//     PlcTask Outputs/Main.M1.Axis.PlcToNc <-> Inputs/FromPlc
//   rixs_optics Instance <-> NC-Task 1 SAF/Axes/M1K2-Yright
//     PlcTask Inputs/Main.M2.Axis.NcToPlc <-> Outputs/ToPlc
//     PlcTask Outputs/Main.M2.Axis.PlcToNc <-> Inputs/FromPlc
//   rixs_optics Instance <-> NC-Task 1 SAF/Axes/M2K2 X
//     PlcTask Inputs/Main.M25.Axis.NcToPlc <-> Outputs/ToPlc
//     PlcTask Outputs/Main.M25.Axis.PlcToNc <-> Inputs/FromPlc
//   rixs_optics Instance <-> NC-Task 1 SAF/Axes/M2K2 Y
//     PlcTask Inputs/Main.M26.Axis.NcToPlc <-> Outputs/ToPlc
//     PlcTask Outputs/Main.M26.Axis.PlcToNc <-> Inputs/FromPlc
//   rixs_optics Instance <-> NC-Task 1 SAF/Axes/M2K2 rX
//     PlcTask Inputs/Main.M27.Axis.NcToPlc <-> Outputs/ToPlc
//     PlcTask Outputs/Main.M27.Axis.PlcToNc <-> Inputs/FromPlc
//   rixs_optics Instance <-> NC-Task 1 SAF/Axes/M3K2 X
//     PlcTask Inputs/Main.M28.Axis.NcToPlc <-> Outputs/ToPlc
//     PlcTask Outputs/Main.M28.Axis.PlcToNc <-> Inputs/FromPlc
//   rixs_optics Instance <-> NC-Task 1 SAF/Axes/M3K2 Y
//     PlcTask Inputs/Main.M29.Axis.NcToPlc <-> Outputs/ToPlc
//     PlcTask Outputs/Main.M29.Axis.PlcToNc <-> Inputs/FromPlc
//   rixs_optics Instance <-> NC-Task 1 SAF/Axes/M3K2 rY
//     PlcTask Inputs/Main.M30.Axis.NcToPlc <-> Outputs/ToPlc
//     PlcTask Outputs/Main.M30.Axis.PlcToNc <-> Inputs/FromPlc
//   rixs_optics Instance <-> NC-Task 1 SAF/Axes/M3K2-BEND-DS
//     PlcTask Inputs/Main.M32.Axis.NcToPlc <-> Outputs/ToPlc
//     PlcTask Outputs/Main.M32.Axis.PlcToNc <-> Inputs/FromPlc
//   rixs_optics Instance <-> NC-Task 1 SAF/Axes/M3K2-BEND-US
//     PlcTask Inputs/Main.M31.Axis.NcToPlc <-> Outputs/ToPlc
//     PlcTask Outputs/Main.M31.Axis.PlcToNc <-> Inputs/FromPlc
//   rixs_optics Instance <-> NC-Task 1 SAF/Axes/M4K2 X
//     PlcTask Inputs/Main.M33.Axis.NcToPlc <-> Outputs/ToPlc
//     PlcTask Outputs/Main.M33.Axis.PlcToNc <-> Inputs/FromPlc
//   rixs_optics Instance <-> NC-Task 1 SAF/Axes/M4K2 Y
//     PlcTask Inputs/Main.M34.Axis.NcToPlc <-> Outputs/ToPlc
//     PlcTask Outputs/Main.M34.Axis.PlcToNc <-> Inputs/FromPlc
//   rixs_optics Instance <-> NC-Task 1 SAF/Axes/M4K2 rX
//     PlcTask Inputs/Main.M35.Axis.NcToPlc <-> Outputs/ToPlc
//     PlcTask Outputs/Main.M35.Axis.PlcToNc <-> Inputs/FromPlc
//   rixs_optics Instance <-> NC-Task 1 SAF/Axes/M4K2-BEND-DS
//     PlcTask Inputs/Main.M37.Axis.NcToPlc <-> Outputs/ToPlc
//     PlcTask Outputs/Main.M37.Axis.PlcToNc <-> Inputs/FromPlc
//   rixs_optics Instance <-> NC-Task 1 SAF/Axes/M4K2-BEND-US
//     PlcTask Inputs/Main.M36.Axis.NcToPlc <-> Outputs/ToPlc
//     PlcTask Outputs/Main.M36.Axis.PlcToNc <-> Inputs/FromPlc
//   rixs_optics Instance <-> NC-Task 1 SAF/Axes/SL1K2-CrystalGap-M22
//     PlcTask Inputs/Main.M22.Axis.NcToPlc <-> Outputs/ToPlc
//     PlcTask Outputs/Main.M22.Axis.PlcToNc <-> Inputs/FromPlc
//   rixs_optics Instance <-> NC-Task 1 SAF/Axes/SL1K2-Pitch-M19
//     PlcTask Inputs/Main.M19.Axis.NcToPlc <-> Outputs/ToPlc
//     PlcTask Outputs/Main.M19.Axis.PlcToNc <-> Inputs/FromPlc
//   rixs_optics Instance <-> NC-Task 1 SAF/Axes/SL1K2-Roll-M21
//     PlcTask Inputs/Main.M21.Axis.NcToPlc <-> Outputs/ToPlc
//     PlcTask Outputs/Main.M21.Axis.PlcToNc <-> Inputs/FromPlc
//   rixs_optics Instance <-> NC-Task 1 SAF/Axes/SL1K2-Vert-M20
//     PlcTask Inputs/Main.M20.Axis.NcToPlc <-> Outputs/ToPlc
//     PlcTask Outputs/Main.M20.Axis.PlcToNc <-> Inputs/FromPlc
//   rixs_optics Instance <-> NC-Task 1 SAF/Axes/SL1K2-YAG-M23
//     PlcTask Inputs/Main.M23.Axis.NcToPlc <-> Outputs/ToPlc
//     PlcTask Outputs/Main.M23.Axis.PlcToNc <-> Inputs/FromPlc
//   rixs_optics Instance <-> NC-Task 1 SAF/Axes/g_h
//     PlcTask Inputs/Main.M9.Axis.NcToPlc <-> Outputs/ToPlc
//     PlcTask Outputs/Main.M9.Axis.PlcToNc <-> Inputs/FromPlc
//   rixs_optics Instance <-> NC-Task 1 SAF/Axes/g_pi
//     PlcTask Outputs/Main.M7.Axis.PlcToNc <-> Inputs/FromPlc
//     StatsTask Inputs/Main.M7.Axis.NcToPlc <-> Outputs/ToPlc
//   rixs_optics Instance <-> NC-Task 1 SAF/Axes/m_h
//     PlcTask Inputs/Main.M8.Axis.NcToPlc <-> Outputs/ToPlc
//     PlcTask Outputs/Main.M8.Axis.PlcToNc <-> Inputs/FromPlc
//   rixs_optics Instance <-> NC-Task 1 SAF/Axes/m_pi
//     PlcTask Outputs/Main.M6.Axis.PlcToNc <-> Inputs/FromPlc
//     StatsTask Inputs/Main.M6.Axis.NcToPlc <-> Outputs/ToPlc
//   rixs_optics Instance <-> NC-Task 1 SAF/Axes/s_io
//     PlcTask Inputs/Main.M10.Axis.NcToPlc <-> Outputs/ToPlc
//     PlcTask Outputs/Main.M10.Axis.PlcToNc <-> Inputs/FromPlc
//   rixs_optics Instance <-> NC-Task 1 SAF/Axes/s_r
//     PlcTask Inputs/Main.M11.Axis.NcToPlc <-> Outputs/ToPlc
//     PlcTask Outputs/Main.M11.Axis.PlcToNc <-> Inputs/FromPlc

CONFIGURATION rixs_optics
    RESOURCE PLC ON TwinCAT3
        TASK DaqTask(INTERVAL := T#1ms, PRIORITY := 19);
        TASK PiezoDriver(INTERVAL := T#1ms, PRIORITY := 3);
        TASK PlcTask(INTERVAL := T#10ms, PRIORITY := 20);
        TASK SerialIO(INTERVAL := T#2ms, PRIORITY := 1);
        TASK StatsTask(INTERVAL := T#2ms, PRIORITY := 2);
        PROGRAM PRG_DAQ_ENCODER WITH DaqTask : PRG_DAQ_ENCODER;
        PROGRAM PiezoSerial WITH PiezoDriver : PiezoSerial;
        PROGRAM PRG_1_PlcTask WITH PlcTask : PRG_1_PlcTask;
        PROGRAM P_Serial_Com WITH SerialIO : P_Serial_Com;
        PROGRAM PRG_Stats WITH StatsTask : PRG_Stats;
    END_RESOURCE
END_CONFIGURATION

// ---- DUTs/ENUM_XS_YAG_States.TcDUT
{attribute 'qualified_only'}
TYPE ENUM_XS_YAG_States :
(
    Unknown := 0,
    OUT := 1,
    YAG1 := 2,
    YAG2 := 3
);
END_TYPE

// ---- DUTs/E_B4C_Rh_CoatingStates.TcDUT
{attribute 'qualified_only'}
{attribute 'strict'}
TYPE E_B4C_Rh_CoatingStates :
(
    Unknown := 0,
    B4C := 1,
    Rh := 2
) UINT;
END_TYPE

// ---- DUTs/E_MR1K1_States.TcDUT
{attribute 'qualified_only'}
{attribute 'strict'}
TYPE E_MR1K1_States :
(
    Unknown := 0,
    B4C := 1,
    OUT := 2
) UINT;
END_TYPE

// ---- DUTs/E_Grating_States.TcDUT
{attribute 'qualified_only'}
{attribute 'strict'}
TYPE E_Grating_States :
(
    Unknown := 0,
    LRG := 1,
    Unruled := 2,
    YAG := 3,
    MEG := 4,
    HEG := 5,
    LEG := 6
) UINT;
END_TYPE

// ---- POUs/DAQ Comm/DUT_01_Channel_NW.TcDUT
TYPE DUT_01_Channel_NW :
STRUCT
    header: DUT_Header_NW;
    channel1: DUT_Channel_NW;
END_STRUCT
END_TYPE

// ---- POUs/DAQ Comm/DUT_Channel_NW.TcDUT
TYPE DUT_Channel_NW :
STRUCT
    count: DWORD;                       // 4    4
    timing: DWORD;                      // 4    8
    scale: WORD;                        // 2    10
    hardwareID: ARRAY [0..15] OF BYTE;  // 16   26
    reserved1: BYTE;                    // 1    27
    channel: BYTE;                      // 1    28
    error: BYTE;                        // 1    29
    mode: BYTE;                         // 1    30
    scale_denominator: WORD;            // 2    32
END_STRUCT
END_TYPE
(*
typedef struct {
    uint32_t    encoderValue;       // network byte order
    uint32_t    timing;             // network byte order
    uint16_t    scale;              // network byte order
    char        hardwareID[16];
    uint8_t     reserved1;
    uint8_t     channel;
    uint8_t     error;
    uint8_t     mode;
    uint16_t     scale_denominator; // network byte order
} encoder_channel_t;
*)

// ---- POUs/DAQ Comm/DUT_Header_NW.TcDUT
TYPE DUT_Header_NW :
STRUCT
    frameCount: WORD;                   // 2    2
    reserved1: WORD;                    // 2    4
    major: WORD;                        // 2    6
    minor: BYTE;                        // 1    7
    micro: BYTE;                        // 1    8
    hardwareID: ARRAY [0..15] OF BYTE;  // 16   24
    reserved2: BYTE;                    // 1    25
    channelMask: BYTE;                  // 1    26
    errorMask: BYTE;                    // 1    27
    mode: BYTE;                         // 1    28
    reserved3: DWORD;                   // 4    32
END_STRUCT
END_TYPE
(*
typedef struct {
    uint16_t    frameCount;         // network byte order
    uint8_t     reserved1[2];
    uint16_t    majorVersion;       // network byte order
    uint8_t     minorVersion;
    uint8_t     microVersion;
    char        hardwareID[16];
    uint8_t     reserved2;
    uint8_t     channelMask;
    uint8_t     errorMask;
    uint8_t     mode;
    uint8_t     reserved3[4];
} encoder_header_t;
*)

// ---- Version/Global_Version.TcGVL
{attribute 'TcGenerated'}
{attribute 'no-analysis'}
{attribute 'linkalways'}
// This function has been automatically generated from the project information.
VAR_GLOBAL CONSTANT
    {attribute 'const_non_replaced'}
    stLibVersion_rix_optics : ST_LibVersion := (iMajor := 3, iMinor := 10, iBuild := 0, iRevision := 0, nFlags := 1, sVersion := '3.10.0');
END_VAR

// ---- GVLs/GVL_COM_Buffers.TcGVL
VAR_GLOBAL
    // M1K2
    Serial_RXBuffer_M1K2 : ComBuffer;
    Serial_TXBuffer_M1K2 : ComBuffer;
END_VAR

// ---- GVLs/GVL_M1K1.TcGVL
{attribute 'qualified_only'}
VAR_GLOBAL
    // Pitch Mechanism:\
    // Currently unused
    {attribute 'TcLinkTo' := '.diEncCnt:=TIIB[EL5042_M1K2_Pitch]^FB Inputs Channel 1^Position'}
    M1K1_Pitch : HOMS_PitchMechanism := (ReqPosLimHi := 24681,
                                         ReqPosLimLo := 24321,
                                         diEncPosLimHi := 10139808,
                                         diEncPosLimLo := 9950984); // Set to 50 urad before hard limits tripped during SAT
END_VAR

// ---- GVLs/GVL_M1K1_BENDER_Constants.TcGVL
{attribute 'qualified_only'}
VAR_GLOBAL CONSTANT
    // Encoder reference values in counts = nm
    nM1K1bendUS_ENC_REF : ULINT := 21458400;
    nM1K1bendDS_ENC_REF : ULINT := 21225900;

    // PMPS Limits for benders
    nM1K1bendUS_PMPS_UpperLimit : ULINT := 22100000; //21500000;//22100000; As requested by Alex R and RP, switched back again
    nM1K1bendUS_PMPS_LowerLimit : ULINT := 20900000; //20100000;//20900000;

    nM1K1bendDS_PMPS_UpperLimit : ULINT := 21800000;//21100000;//21800000;
    nM1K1bendDS_PMPS_LowerLimit : ULINT := 20600000;// 19800000;//20600000;
END_VAR

// ---- GVLs/GVL_M1K1_BENDER_RTD.TcGVL
{attribute 'qualified_only'}
VAR_GLOBAL
    // M1K1 US RTDs
    {attribute 'TcLinkTo' := 'TIIB[EL3202-0010_M1K1US1_M1K1US2]^RTD Inputs Channel 1^Value'}
    nM1K1US_RTD_1 AT %I* : INT;
    {attribute 'TcLinkTo' := 'TIIB[EL3202-0010_M1K1US1_M1K1US2]^RTD Inputs Channel 2^Value'}
    nM1K1US_RTD_2 AT %I* : INT;
    {attribute 'TcLinkTo' := 'TIIB[EL3202-0010_M1K1US3_M1K1DS1]^RTD Inputs Channel 1^Value'}
    nM1K1US_RTD_3 AT %I* : INT;

    // M1K1 DS RTDs
    {attribute 'TcLinkTo' := 'TIIB[EL3202-0010_M1K1US3_M1K1DS1]^RTD Inputs Channel 2^Value'}
    nM1K1DS_RTD_1 AT %I* : INT;
    {attribute 'TcLinkTo' := 'TIIB[EL3202-0010_M1K1DS2_M1K1DS3]^RTD Inputs Channel 1^Value'}
    nM1K1DS_RTD_2 AT %I* : INT;
    {attribute 'TcLinkTo' := 'TIIB[EL3202-0010_M1K1DS2_M1K1DS3]^RTD Inputs Channel 2^Value'}
    nM1K1DS_RTD_3 AT %I* : INT;

END_VAR

// ---- GVLs/GVL_M1K1_Constants.TcGVL
{attribute 'qualified_only'}
VAR_GLOBAL CONSTANT
    // Encoder reference values in counts = nm
    // Enc reference values from Axilon FAT
    nYUP_ENC_REF : ULINT := 13008545;
    nYDWN_ENC_REF : ULINT := 11158257;
    nXUP_ENC_REF : ULINT := 19831295;
    nXDWN_ENC_REF : ULINT := 19604132;

    (* previous values
    nXUP_ENC_REF : ULINT := 19649910;
    nXDWN_ENC_REF : ULINT := 19609100;
    *)
END_VAR

// ---- GVLs/GVL_M1K2.TcGVL
{attribute 'qualified_only'}
VAR_GLOBAL
    // Pitch Mechanism:
    // Currently Unused
    {attribute 'TcLinkTo' := '.diEncCnt:=TIIB[EL5042_M1K2_Pitch]^FB Inputs Channel 1^Position'}
    M1K2_Pitch : HOMS_PitchMechanism := (ReqPosLimHi := 200,
                                         ReqPosLimLo := -30,
                                         diEncPosLimHi := 10121210,
                                         diEncPosLimLo := 10004610); // Set to 50 urad before hard limits tripped during SAT
END_VAR

// ---- GVLs/GVL_M2K2.TcGVL
{attribute 'qualified_only'}
VAR_GLOBAL CONSTANT
    // Encoder reference values in counts = nm
    // Put encoder reference values for nominal 0 here
    nM2K2X_ENC_REF : ULINT := 6077000; //these numbers
    nM2K2Y_ENC_REF : ULINT := 5975460; //are
    nM2K2rX_ENC_REF : ULINT := 50412360;//real
END_VAR

// ---- GVLs/GVL_M3K2.TcGVL
{attribute 'qualified_only'}
VAR_GLOBAL CONSTANT
    // Encoder reference values in counts = nm
    // Put encoder reference values for nominal 0 here
    nM3K2X_ENC_REF : ULINT := 5951195;
    nM3K2Y_ENC_REF : ULINT := 5857203;
    nM3K2rY_ENC_REF : ULINT := 39991700;
    nM3K2US_ENC_REF : ULINT := 1234567; //these numbers
    nM3K2DS_ENC_REF : ULINT := 1234567;	 //are not real!!

(*
    // PMPS Limits for benders - need to identify these
    nM3K2US_PMPS_UpperLimit : ULINT := 21500000;//22100000;
    nM3K2US_PMPS_LowerLimit : ULINT := 20100000;//20900000;

    nM3K2DS_PMPS_UpperLimit : ULINT := 21100000;//21800000;
    nM3K2DS_PMPS_LowerLimit : ULINT := 19800000;//20600000;
*)
END_VAR

VAR_GLOBAL
    // M3K2 US RTDs
    {attribute 'TcLinkTo' := 'TIIB[EL3202-0010_M3K2US1_M3K2US2]^RTD Inputs Channel 1^Value'}
    nM3K2US_RTD_1 AT %I* : INT;
    {attribute 'TcLinkTo' := 'TIIB[EL3202-0010_M3K2US1_M3K2US2]^RTD Inputs Channel 2^Value'}
    nM3K2US_RTD_2 AT %I* : INT;


    // M3K2 DS RTDs
    {attribute 'TcLinkTo' := 'TIIB[EL3202-0010_M3K2US3_M3K2DS1]^RTD Inputs Channel 2^Value'}
    nM3K2DS_RTD_1 AT %I* : INT;
    {attribute 'TcLinkTo' := 'TIIB[EL3202-0010_M3K2DS2_M3K2DS3]^RTD Inputs Channel 2^Value'}
    nM3K2DS_RTD_3 AT %I* : INT;

END_VAR

// ---- GVLs/GVL_M4K2.TcGVL
{attribute 'qualified_only'}
VAR_GLOBAL CONSTANT
    // Encoder reference values in counts = nm
    // Put encoder reference values for nominal 0 here
    nM4K2X_ENC_REF : ULINT := 5902073;
    nM4K2Y_ENC_REF : ULINT := 6000313;
    nM4K2rX_ENC_REF : ULINT := 50657020;
    nM4K2US_ENC_REF : ULINT := 1234567; //these numbers
    nM4K2DS_ENC_REF : ULINT := 1234567; //are not real!!

    // PMPS Limits for benders - need to identify these
    nM4K2US_PMPS_UpperLimit : ULINT := 21500000;//22100000;
    nM4K2US_PMPS_LowerLimit : ULINT := 20100000;//20900000;

    nM4K2DS_PMPS_UpperLimit : ULINT := 21100000;//21800000;
    nM4K2DS_PMPS_LowerLimit : ULINT := 19800000;//20600000;
END_VAR

VAR_GLOBAL
    // M4K2 US RTDs
    {attribute 'TcLinkTo' := 'TIIB[EL3202-0010_M4K2US1_M4K2US2]^RTD Inputs Channel 1^Value'}
    nM4K2US_RTD_1 AT %I* : INT;
    {attribute 'TcLinkTo' := 'TIIB[EL3202-0010_M4K2US1_M4K2US2]^RTD Inputs Channel 2^Value'}
    nM4K2US_RTD_2 AT %I* : INT;
    {attribute 'TcLinkTo' := 'TIIB[EL3202-0010_M4K2US3_M4K2DS1]^RTD Inputs Channel 1^Value'}
    nM4K2US_RTD_3 AT %I* : INT;

    // M4K2 DS RTDs
    {attribute 'TcLinkTo' := 'TIIB[EL3202-0010_M4K2US3_M4K2DS1]^RTD Inputs Channel 2^Value'}
    nM4K2DS_RTD_1 AT %I* : INT;


END_VAR

// ---- GVLs/GVL_M1K2_Constants.TcGVL
{attribute 'qualified_only'}
VAR_GLOBAL CONSTANT
    // Encoder reference values in counts = nm
    // Enc reference values after alignment 3-13-20
    nYLEFT_ENC_REF : ULINT := 99171678;
    nYRIGHT_ENC_REF : ULINT := 101371326;
    nXUP_ENC_REF : ULINT := 19501048;
    nXDWN_ENC_REF : ULINT := 20872028;

    // Lever arm for Yright/Yleft -> Roll about Z-axis
    fRollLeverArm_um : REAL := 717000; // lever arm for Yright/Yleft axes in um
END_VAR

// ---- GVLs/GVL_PMPS.TcGVL
{attribute 'qualified_only'}
VAR_GLOBAL
    {attribute 'pytmc' := 'pv: PLC:RIX:OPTICS:ARB:01'}
    fbArbiter1: FB_Arbiter(1);
    {attribute 'pytmc' := 'pv: PLC:RIX:OPTICS:ARB:02'}
    fbArbiter2: FB_Arbiter(2);
    {attribute 'pytmc' := 'pv: PLC:RIX:OPTICS:FFO:01'}
    {attribute 'TcLinkTo' := '.q_xFastFaultOut:=TIIB[PMPS_FFO]^Channel 1^Output'}
    fbFastFaultOutput1: FB_HardwareFFOutput := (bAutoReset := TRUE , i_sNetID:='172.21.42.126.1.1' );
    {attribute 'pytmc' := 'pv: PLC:RIX:OPTICS:FFO:02'}
    {attribute 'TcLinkTo' := '.q_xFastFaultOut:=TIIB[PMPS_FFO]^Channel 2^Output'}
    fbFastFaultOutput2: FB_HardwareFFOutput := (bAutoReset := TRUE, i_sNetID:='172.21.42.126.1.1');
    rPhotonEnergy: REAL;
END_VAR

// ---- GVLs/GVL_SerialIO.TcGVL
VAR_GLOBAL
    //Better have your inputs and outputs!
    // M1K2
    Serial_stComIn_M1K2   AT %I*	:	EL6inData22B (*KL6inData22B*);
    Serial_stComOut_M1K2  AT %Q*	:	EL6outData22B (*KL6outData22B*);
END_VAR

// ---- GVLs/GVL_States.TcGVL
{attribute 'qualified_only'}
VAR_GLOBAL
    stDefaultOffsetY : ST_PositionState := (
        fDelta:=2000,
        fVelocity:=100,
        fAccel:=5050,
        fDecel:=5050,
        bMoveOk:=TRUE,
        bValid:=TRUE,
        bUseRawCounts:=TRUE
    );
        stDefaultOffsetX : ST_PositionState := (
        fDelta:=10000,
        fVelocity:=150,
        fAccel:=1000,
        fDecel:=1000,
        bMoveOk:=TRUE,
        bValid:=TRUE,
        bUseRawCounts:=TRUE
    );
        stDefaultKBX : ST_PositionState := (
        fDelta:=5,
        fVelocity:=0.3,
        fAccel:=100,
        fDecel:=100,
        bMoveOk:=TRUE,
        bValid:=TRUE,
        bUseRawCounts:=TRUE
    );
        stDefaultKBY : ST_PositionState := (
        fDelta:=5,
        fVelocity:=0.3,
        fAccel:=10,
        fDecel:=10,
        bMoveOk:=TRUE,
        bValid:=TRUE,
        bUseRawCounts:=TRUE
    );
END_VAR

// ---- GVLs/Main.TcGVL
VAR_GLOBAL
(*
    Only includes motor definitions for the IOC
    These are hard-coded to be Main.M#,
    but are very convenient to store in a GVL,
    hence the confusing namespace here

    This should be refactored once the IOC
    supports arbitrary ads paths for motors
*)
    (*MR1K2*)
    // Motors
    {attribute 'TcLinkTo' := '.bLimitForwardEnable:=TIIB[EL7047_M1K2_Yleft]^STM Status^Status^Digital input 1;
                              .bLimitBackwardEnable:=TIIB[EL7047_M1K2_Yleft]^STM Status^Status^Digital input 2;
                              .nRawEncoderULINT:=TIIB[EL5042_M1K2_Yleftright]^FB Inputs Channel 1^Position'}
    {attribute 'pytmc' := '
        pv: MR1K2:SWITCH:MMS:YLEFT
    '}
    M1 : ST_MotionStage := (fVelocity:=100.0, nEnableMode:=ENUM_StageEnableMode.ALWAYS, bPowerSelf:=False); // M1K2 Yleft
    fbMotionStage_m1 : FB_MotionStage;

    {attribute 'TcLinkTo' := '.bLimitForwardEnable:=TIIB[EL7047_M1K2_Yright]^STM Status^Status^Digital input 1;
                              .bLimitBackwardEnable:=TIIB[EL7047_M1K2_Yright]^STM Status^Status^Digital input 2;
                              .nRawEncoderULINT:=TIIB[EL5042_M1K2_Yleftright]^FB Inputs Channel 2^Position'}
    {attribute 'pytmc' := '
        pv: MR1K2:SWITCH:MMS:YRIGHT
    '}
    M2 : ST_MotionStage := (fVelocity:=100.0, nEnableMode:=ENUM_StageEnableMode.ALWAYS, bPowerSelf:=True); // M1K2 Yright
    fbMotionStage_m2 : FB_MotionStage;
    {attribute 'TcLinkTo' := '.bLimitForwardEnable:=TIIB[EL7047_M1K2_Xup]^STM Status^Status^Digital input 1;
                              .bLimitBackwardEnable:=TIIB[EL7047_M1K2_Xup]^STM Status^Status^Digital input 2;
                               .nRawEncoderULINT:=TIIB[EL5042_M1K2_Xupdwn]^FB Inputs Channel 1^Position'}
    {attribute 'pytmc' := '
        pv: MR1K2:SWITCH:MMS:XUP
    '}
    M3 : ST_MotionStage := (fVelocity:=150.0, nEnableMode:=ENUM_StageEnableMode.ALWAYS, bPowerSelf:=True); // M1K2 Xup
    fbMotionStage_m3 : FB_MotionStage;

    {attribute 'TcLinkTo' := '.bLimitForwardEnable:=TIIB[EL7047_M1K2_Xdwn]^STM Status^Status^Digital input 1;
                              .bLimitBackwardEnable:=TIIB[EL7047_M1K2_Xdwn]^STM Status^Status^Digital input 2;
                              .nRawEncoderULINT:=TIIB[EL5042_M1K2_Xupdwn]^FB Inputs Channel 1^Position'}
    {attribute 'pytmc' := '
        pv: MR1K2:SWITCH:MMS:XDWN
    '}
    M4 : ST_MotionStage := (fVelocity:=150.0, nEnableMode:=ENUM_StageEnableMode.ALWAYS, bPowerSelf:=True); // M1K2 Xdwn
    fbMotionStage_m4 : FB_MotionStage;

    {attribute 'TcLinkTo' := '.bLimitForwardEnable:=TIIB[EL7047_M1K2_PitchCoarse]^STM Status^Status^Digital input 1;
                              .bLimitBackwardEnable:=TIIB[EL7047_M1K2_PitchCoarse]^STM Status^Status^Digital input 2;
                              .nRawEncoderULINT:=TIIB[EL5042_M1K2_Pitch]^FB Inputs Channel 1^Position'}
    {attribute 'pytmc' := '
        pv: MR1K2:SWITCH:MMS:PITCH
    '}
    M5 : ST_MotionStage := (fVelocity:=30.0, nEnableMode:=ENUM_StageEnableMode.DURING_MOTION, bPowerSelf:=True); // M1K2 Pitch Stepper


    (*SP1K1-Mono*)
    {attribute 'pytmc' := '
        pv: SP1K1:MONO:MMS:M_PI
    '}
    {attribute 'TcLinkTo' := '.bLimitForwardEnable:=TIIB[m_pi_m]^STM Status^Status^Digital input 1;
                              .bLimitBackwardEnable:=TIIB[m_pi_m]^STM Status^Status^Digital input 2;
                              .nRawEncoderULINT:=TIIB[m_pi_up_dwn_e]^FB Inputs Channel 2^Position'}
    M6: ST_MotionStage:=(nEnableMode:=ENUM_StageEnableMode.ALWAYS, fVelocity:=200.0, bPowerSelf:=True); // M_PI, urad
    {attribute 'pytmc' := '
        pv: SP1K1:MONO:MMS:G_PI
    '}
    {attribute 'TcLinkTo' := '.bLimitForwardEnable:=TIIB[g_pi_m]^STM Status^Status^Digital input 1;
                              .bLimitBackwardEnable:=TIIB[g_pi_m]^STM Status^Status^Digital input 2;
                              .nRawEncoderULINT:=TIIB[g_pi_up_dwn_e]^FB Inputs Channel 1^Position'}
    M7: ST_MotionStage:=(nEnableMode:=ENUM_StageEnableMode.ALWAYS, fVelocity:=200.0, bPowerSelf:=True); // G_PI, urad
    {attribute 'pytmc' := '
        pv: SP1K1:MONO:MMS:M_H
    '}
    {attribute 'TcLinkTo' := '.bLimitForwardEnable:=TIIB[m_h_m]^STM Status^Status^Digital input 1;
                              .bLimitBackwardEnable:=TIIB[m_h_m]^STM Status^Status^Digital input 2;
                              .nRawEncoderULINT:=TIIB[m_h_e-g_h_e]^FB Inputs Channel 1^Position'}
    M8: ST_MotionStage:=(nEnableMode:=ENUM_StageEnableMode.DURING_MOTION, fVelocity:=500.0, bPowerSelf:=True); // M_H, um
    {attribute 'pytmc' := '
        pv: SP1K1:MONO:MMS:G_H
    '}
    {attribute 'TcLinkTo' := '.bLimitForwardEnable:=TIIB[g_h_m]^STM Status^Status^Digital input 1;
                              .bLimitBackwardEnable:=TIIB[g_h_m]^STM Status^Status^Digital input 2;
                              .nRawEncoderULINT:=TIIB[m_h_e-g_h_e]^FB Inputs Channel 2^Position'}
    M9: ST_MotionStage:=(nEnableMode:=ENUM_StageEnableMode.DURING_MOTION, fVelocity:=1000.0, bPowerSelf:=False); // G_H, um
    {attribute 'pytmc' := '
        pv: SP1K1:MONO:MMS:SD_V
    '}
    {attribute 'TcLinkTo' := '.bLimitForwardEnable:=TIIB[s_io_m]^STM Status^Status^Digital input 1;
                              .bLimitBackwardEnable:=TIIB[s_io_m]^STM Status^Status^Digital input 2'}
    M10: ST_MotionStage:=(nEnableMode:=ENUM_StageEnableMode.DURING_MOTION, fVelocity:=500.0, bPowerSelf:=True); // SD_V, um
    {attribute 'pytmc' := '
        pv: SP1K1:MONO:MMS:SD_ROT
    '}
    // no limits on this motion
    M11: ST_MotionStage:=(nEnableMode:=ENUM_StageEnableMode.DURING_MOTION, fVelocity:=500.0, bPowerSelf:=True); // SD_R, urad

    (*MR1K1*)
    // Should move before MR1K2 and re-number each motor, lots of work
    // need to fix Axis IDs for IOC to work
    // For now just want functional PLC project
    // Motors

    {attribute 'TcLinkTo' := '.bLimitBackwardEnable:=TIIB[EL7047_M1K1_Ydwn]^STM Status^Status^Digital input 2;
                              .bLimitForwardEnable:=TIIB[EL7047_M1K1_Ydwn]^STM Status^Status^Digital input 1;
                              .nRawEncoderULINT:=TIIB[EL5042_M1K1_Yupdwn]^FB Inputs Channel 1^Position'}
    {attribute 'pytmc' := '
        pv: MR1K1:BEND:MMS:YUP
    '}
    M12 : ST_MotionStage := (fVelocity:=100.0, nEnableMode:=ENUM_StageEnableMode.ALWAYS, bPowerSelf:=False); // M1K1 Yup
    fbMotionStage_m12 : FB_MotionStage;
    {attribute 'TcLinkTo' := '.bLimitForwardEnable:=TIIB[EL7047_M1K1_Ydwn]^STM Status^Status^Digital input 1;
                        .bLimitBackwardEnable:=TIIB[EL7047_M1K1_Ydwn]^STM Status^Status^Digital input 2'}
    {attribute 'pytmc' := '
        pv: MR1K1:BEND:MMS:YDWN
    '}
    M13 : ST_MotionStage := (fVelocity:=100.0, nEnableMode:=ENUM_StageEnableMode.ALWAYS, bPowerSelf:=True); // M1K1 Ydwn
    fbMotionStage_m13 : FB_MotionStage;

    {attribute 'TcLinkTo' := '.bLimitForwardEnable:=TIIB[EL7047_M1K1_Xup]^STM Status^Status^Digital input 1;
                              .bLimitBackwardEnable:=TIIB[EL7047_M1K1_Xup]^STM Status^Status^Digital input 2;
                              .nRawEncoderULINT:=TIIB[EL5042_M1K1_Xupdwn]^FB Inputs Channel 1^Position'}
    {attribute 'pytmc' := '
        pv: MR1K1:BEND:MMS:XUP
    '}
    M14 : ST_MotionStage := (fVelocity:=150.0, nEnableMode:=ENUM_StageEnableMode.ALWAYS, bPowerSelf:=False); // M1K1 Xup
    fbMotionStage_m14 : FB_MotionStage;

    {attribute 'TcLinkTo' := '.bLimitForwardEnable:=TIIB[EL7047_M1K1_Xdwn]^STM Status^Status^Digital input 1;
                              .bLimitBackwardEnable:=TIIB[EL7047_M1K1_Xdwn]^STM Status^Status^Digital input 2'}
    {attribute 'pytmc' := '
        pv: MR1K1:BEND:MMS:XDWN
    '}
    M15 : ST_MotionStage := (fVelocity:=150.0, nEnableMode:=ENUM_StageEnableMode.ALWAYS, bPowerSelf:=True); // M1K1 Xdwn
    fbMotionStage_m15 : FB_MotionStage;

    {attribute 'TcLinkTo' := '.bLimitForwardEnable:=TIIB[EL7047_M1K1_PitchCoarse]^STM Status^Status^Digital input 1;
                              .bLimitBackwardEnable:=TIIB[EL7047_M1K1_PitchCoarse]^STM Status^Status^Digital input 2;
                              .nRawEncoderULINT:=TIIB[EL5042_M1K1_Pitch]^FB Inputs Channel 1^Position'}
    {attribute 'pytmc' := '
        pv: MR1K1:BEND:MMS:PITCH
    '}
    M16 : ST_MotionStage := (fVelocity:=30.0, nEnableMode:=ENUM_StageEnableMode.ALWAYS, bPowerSelf:=True); // M1K1 Pitch Stepper

    {attribute 'TcLinkTo' := '.bLimitBackwardEnable:=TIIB[EL7041_M1K1_BEND_US]^STM Status^Status^Digital input 2;
                              .nRawEncoderULINT    := TIIB[EL5042_M1K1_BEND_USDS]^FB Inputs Channel 1^Position'}
    {attribute 'pytmc' := '
    pv: MR1K1:BEND:MMS:US
    '}
    // unlinking this .bLimitForwardEnable :=TIIB[EL7041_M1K1_BEND_US]^STM Status^Status^Digital input 1;
    M17 : ST_MotionStage := (nEnableMode:=ENUM_StageEnableMode.DURING_MOTION, bPowerSelf:=TRUE); //MR1K1 US BEND
    fbMotionStage_m17 : FB_MotionStage;

    {attribute 'TcLinkTo' := '.bLimitForwardEnable :=TIIB[EL7041_M1K1_BEND_DS]^STM Status^Status^Digital input 1;
                              .bLimitBackwardEnable:=TIIB[EL7041_M1K1_BEND_DS]^STM Status^Status^Digital input 2;
                              .nRawEncoderULINT    := TIIB[EL5042_M1K1_BEND_USDS]^FB Inputs Channel 2^Position'}
    {attribute 'pytmc' := '
    pv: MR1K1:BEND:MMS:DS
    '}
    M18 : ST_MotionStage := (nEnableMode:=ENUM_StageEnableMode.DURING_MOTION, bPowerSelf:=TRUE); //MR1K1 DS BEND
    fbMotionStage_m18 : FB_MotionStage;

    (*SL1K2*)
    // Motors
    {attribute 'TcLinkTo' := '.bLimitForwardEnable:=TIIB[EL7047_SL1K2_PITCH]^STM Status^Status^Digital input 2;
                              .bLimitBackwardEnable:=TIIB[EL7047_SL1K2_PITCH]^STM Status^Status^Digital input 1;
                               .nRawEncoderULINT      := TIIB[EL5042_SL1K2_PITCH_VERT]^FB Inputs Channel 1^Position'}
    {attribute 'pytmc' := '
        pv: SL1K2:EXIT:MMS:PITCH
    '}
    M19 : ST_MotionStage := (sName:= 'SL1K2:EXIT:MMS:PITCH',fVelocity :=0.12);// Air Pitch

    {attribute 'TcLinkTo' := '.bLimitForwardEnable:=TIIB[EL7047_SL1K2_VERT]^STM Status^Status^Digital input 1;
                              .bLimitBackwardEnable:=TIIB[EL7047_SL1K2_VERT]^STM Status^Status^Digital input 2;
                               .nRawEncoderULINT      := TIIB[EL5042_SL1K2_PITCH_VERT]^FB Inputs Channel 2^Position'}
    {attribute 'pytmc' := '
        pv: SL1K2:EXIT:MMS:VERT
    '}
    M20 : ST_MotionStage := (sName:= 'SL1K2:EXIT:MMS:VERT',fVelocity :=0.3); // Air Vertical

    {attribute 'TcLinkTo' := '.bLimitForwardEnable:=TIIB[EL7047_SL1K2_ROLL]^STM Status^Status^Digital input 2;
                              .bLimitBackwardEnable:=TIIB[EL7047_SL1K2_ROLL]^STM Status^Status^Digital input 1;
                              .nRawEncoderULINT      := TIIB[EL5042_SL1K2_ROLL_GAP]^FB Inputs Channel 1^Position'}
    {attribute 'pytmc' := '
        pv: SL1K2:EXIT:MMS:ROLL
    '}
    M21 : ST_MotionStage := (sName:= 'SL1K2:EXIT:MMS:ROLL',fVelocity :=0.24); // Air Roll

    {attribute 'TcLinkTo' := '.bLimitForwardEnable:=TIIB[EL7047_SL1K2_GAP]^STM Status^Status^Digital input 1;
                              .bLimitBackwardEnable:=TIIB[EL7047_SL1K2_GAP]^STM Status^Status^Digital input 2;
                              .nRawEncoderULINT      := TIIB[EL5042_SL1K2_ROLL_GAP]^FB Inputs Channel 2^Position'}
    {attribute 'pytmc' := '
        pv: SL1K2:EXIT:MMS:GAP
    '}
    M22 : ST_MotionStage := (sName:= 'SL1K2:EXIT:MMS:GAP',fVelocity :=0.1); // GAP

    {attribute 'TcLinkTo' := '.bLimitForwardEnable:=TIIB[EL7047_SL1K2_YAG]^STM Status^Status^Digital input 2;
                              .bLimitBackwardEnable:=TIIB[EL7047_SL1K2_YAG]^STM Status^Status^Digital input 1;
                              .nRawEncoderULINT      := TIIB[EL5042_SL1K2_YAG]^FB Inputs Channel 1^Position'}
    {attribute 'pytmc' := '
        pv: SL1K2:EXIT:MMS:YAG
    '}
    M23 : ST_MotionStage := (sName:= 'SL1K2:EXIT:MMS:YAG',fVelocity :=0.5); // YAG


    // ST1K1-ZOS-MMS
    {attribute 'pytmc' := 'pv: ST1K1:ZOS:MMS'}
    {attribute 'TcLinkTo' := '.bLimitForwardEnable  := TIIB[ST1K1-EL7041]^STM Status^Status^Digital input 1;
                              .bLimitBackwardEnable := TIIB[ST1K1-EL7041]^STM Status^Status^Digital input 2;
                              .nRawEncoderULINT     :=TIIB[ST1K1-EL5042]^FB Inputs Channel 1^Position;
                              .bBrakeRelease        := TIIB[ST1K1-EL2008]^Channel 1^Output'}
    M24: ST_MotionStage := (sName := 'ST1K1:ZOS:MMS');

    // MR2K2-FLAT axes
    {attribute 'pytmc' := 'pv: MR2K2:FLAT:MMS:X'}
    {attribute 'TcLinkTo' := '.bLimitForwardEnable:=TIIB[EL7041_M2K2X]^STM Status^Status^Digital input 1;
                              .bLimitBackwardEnable:=TIIB[EL7041_M2K2X]^STM Status^Status^Digital input 2;
                              .nRawEncoderULINT:=TIIB[EL5042_M2K2X_M2K2Y]^FB Inputs Channel 1^Position'}
    M25 : ST_MotionStage := (nEnableMode:=ENUM_StageEnableMode.ALWAYS, bPowerSelf:=FALSE); //X mot
       fbMotionStageM25 : FB_MotionStage;
    {attribute 'pytmc' := 'pv: MR2K2:FLAT:MMS:Y'}
    {attribute 'TcLinkTo' := '.bLimitForwardEnable:=TIIB[EL7041_M2K2Y]^STM Status^Status^Digital input 1;
                              .bLimitBackwardEnable:=TIIB[EL7041_M2K2Y]^STM Status^Status^Digital input 2;
                              .nRawEncoderULINT:=TIIB[EL5042_M2K2X_M2K2Y]^FB Inputs Channel 2^Position'}
    M26 : ST_MotionStage := (nEnableMode:=ENUM_StageEnableMode.ALWAYS, bPowerSelf:=TRUE); //Y mot
    fbMotionStageM26 : FB_MotionStage;
    {attribute 'pytmc' := 'pv: MR2K2:FLAT:MMS:PITCH'}
    {attribute 'TcLinkTo' := '.bLimitForwardEnable:=TIIB[EL7041_M2K2rX]^STM Status^Status^Digital input 2;
                              .bLimitBackwardEnable:=TIIB[EL7041_M2K2rX]^STM Status^Status^Digital input 1;
                              .nRawEncoderULINT:=TIIB[EL5042_M2K2rX]^FB Inputs Channel 1^Position'}
    M27 : ST_MotionStage := (nEnableMode:=ENUM_StageEnableMode.ALWAYS, bPowerSelf:=TRUE); //Pitch mot
    fbMotionStageM27 : FB_MotionStage;

    // MR3K2-KBH axes
    {attribute 'pytmc' := 'pv: MR3K2:KBH:MMS:X'}
    {attribute 'TcLinkTo' := '.bLimitForwardEnable:=TIIB[EL7041_M3K2X]^STM Status^Status^Digital input 1;
                              .bLimitBackwardEnable:=TIIB[EL7041_M3K2X]^STM Status^Status^Digital input 2;
                              .nRawEncoderULINT:=TIIB[EL5042_M3K2X_M3K2Y]^FB Inputs Channel 1^Position'}
    M28 : ST_MotionStage := (nEnableMode:=ENUM_StageEnableMode.ALWAYS, bPowerSelf:=TRUE); //X mot
    fbMotionStageM28 : FB_MotionStage;
    {attribute 'pytmc' := 'pv: MR3K2:KBH:MMS:Y'}
    {attribute 'TcLinkTo' := '.bLimitForwardEnable:=TIIB[EL7041_M3K2Y]^STM Status^Status^Digital input 1;
                              .bLimitBackwardEnable:=TIIB[EL7041_M3K2Y]^STM Status^Status^Digital input 2;
                              .nRawEncoderULINT:=TIIB[EL5042_M3K2X_M3K2Y]^FB Inputs Channel 2^Position'}
    M29 : ST_MotionStage := (nEnableMode:=ENUM_StageEnableMode.ALWAYS, bPowerSelf:=FALSE); //Y mot
    fbMotionStageM29 : FB_MotionStage;
    {attribute 'pytmc' := 'pv: MR3K2:KBH:MMS:PITCH'}
    {attribute 'TcLinkTo' := '.bLimitForwardEnable:=TIIB[EL7041_M3K2rY]^STM Status^Status^Digital input 1;
                              .bLimitBackwardEnable:=TIIB[EL7041_M3K2ry]^STM Status^Status^Digital input 2;
                              .nRawEncoderULINT:=TIIB[EL5042_M3K2rY]^FB Inputs Channel 1^Position'}
    M30 : ST_MotionStage := (nEnableMode:=ENUM_StageEnableMode.ALWAYS, bPowerSelf:=TRUE); //Pitch mot
    fbMotionStageM30 : FB_MotionStage;
    {attribute 'pytmc' := '	pv: MR3K2:KBH:MMS:BEND:US'}
    {attribute 'TcLinkTo' := '.bLimitForwardEnable :=TIIB[EL7041_M3K2_BEND_US]^STM Status^Status^Digital input 1;
                              .bLimitBackwardEnable:=TIIB[EL7041_M3K2_BEND_US]^STM Status^Status^Digital input 2;
                              .nRawEncoderULINT:= TIIB[EL5042_M3K2_BEND_USDS]^FB Inputs Channel 1^Position'}
    M31 : ST_MotionStage := (nEnableMode:=ENUM_StageEnableMode.DURING_MOTION, bPowerSelf:=TRUE); //MR3K2 US BEND
    fbMotionStageM31 : FB_MotionStage;
    {attribute 'pytmc' := 'pv: MR3K2:KBH:MMS:BEND:DS'}
    {attribute 'TcLinkTo' := '.bLimitForwardEnable :=TIIB[EL7041_M3K2_BEND_DS]^STM Status^Status^Digital input 1;
                              .bLimitBackwardEnable:=TIIB[EL7041_M3K2_BEND_DS]^STM Status^Status^Digital input 2;
                              .nRawEncoderULINT:= TIIB[EL5042_M3K2_BEND_USDS]^FB Inputs Channel 2^Position'}
    M32 : ST_MotionStage := (nEnableMode:=ENUM_StageEnableMode.DURING_MOTION, bPowerSelf:=TRUE); //MR3K2 DS BEND
    fbMotionStageM32 : FB_MotionStage;


